KUKA KRL program: MyProgram_029().src

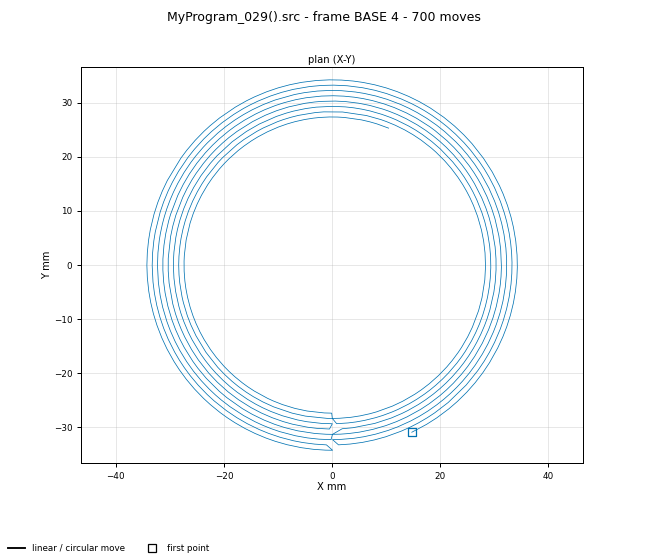
[picture p0: tool path of MyProgram_029().src in frame BASE 4, 700 of 700 moves have a stored position in this frame; points joined in program order, loops and branches not executed]
&ACCESS RVP
&REL 1
&PARAM TEMPLATE = C:\KRC\Roboter\Template\vorgabe
&PARAM EDITMASK = *
DEF MyProgram_029()
; ---- Setting reference (Base) ----
$BASE = BASE_DATA[4]

; --------------------------
; ---- Setting tool (TCP) ----
$TOOL = TOOL_DATA[3]
; --------------------------

$VEL.CP = VEL_APROX_PRINT
Startdeposition()
$VEL.CP = VEL_PRINT
LIN {X 14.7405,Y -30.9266,Z 59,A -69.7461,B 24.853,C -2.7977,E1 25.0726,E2 -567.2107} C_DIS
LIN {X 17.464,Y -29.4746,Z 59,A -65.0615,B 24.8527,C -2.8002,E1 25.084,E2 -571.8873} C_DIS
LIN {X 19.3591,Y -28.2666,Z 59,A -61.3011,B 24.8519,C -2.8074,E1 25.0927,E2 -575.6523} C_DIS
LIN {X 21.5912,Y -26.5997,Z 59,A -56.6338,B 24.8509,C -2.8173,E1 25.103,E2 -580.3259} C_DIS
LIN {X 23.1828,Y -25.2248,Z 59,A -53.0148,B 24.8499,C -2.8266,E1 25.1106,E2 -583.9526} C_DIS
LIN {X 24.9271,Y -23.5028,Z 59,A -49.0912,B 24.8491,C -2.8339,E1 25.1182,E2 -587.8767} C_DIS
LIN {X 26.474,Y -21.7461,Z 59,A -45.15,B 24.848,C -2.8442,E1 25.1254,E2 -591.8243} C_DIS
LIN {X 27.8774,Y -19.9147,Z 59,A -41.382,B 24.8471,C -2.8531,E1 25.1316,E2 -595.5953} C_DIS
LIN {X 29.1256,Y -18.0405,Z 59,A -37.326,B 24.8455,C -2.8677,E1 25.1377,E2 -599.6654} C_DIS
LIN {X 30.6261,Y -15.3561,Z 59,A -32.4503,B 24.8443,C -2.8785,E1 25.1442,E2 -604.541} C_DIS
LIN {X 31.5991,Y -13.2381,Z 59,A -28.9182,B 24.8437,C -2.8846,E1 25.1481,E2 -608.0684} C_DIS
LIN {X 32.2982,Y -11.4269,Z 59,A -25.3896,B 24.8421,C -2.8985,E1 25.1516,E2 -611.6102} C_DIS
LIN {X 32.9807,Y -9.2749,Z 59,A -21.6584,B 24.8409,C -2.9094,E1 25.1545,E2 -615.3459} C_DIS
LIN {X 33.5316,Y -7.0281,Z 59,A -17.8504,B 24.8397,C -2.9205,E1 25.1569,E2 -619.1581} C_DIS
LIN {X 33.9066,Y -4.9084,Z 59,A -14.2291,B 24.8384,C -2.9321,E1 25.1585,E2 -622.7854} C_DIS
LIN {X 34.1715,Y -2.4646,Z 59,A -10.3592,B 24.8374,C -2.9414,E1 25.1595,E2 -626.6544} C_DIS
LIN {X 34.2581,Y -0.4122,Z 59,A -7.0062,B 24.8364,C -2.9509,E1 25.1598,E2 -630.01} C_DIS
LIN {X 34.2094,Y 1.8598,Z 59,A -2.861,B 24.8345,C -2.9678,E1 25.1593,E2 -634.1707} C_DIS
LIN {X 33.9679,Y 4.4635,Z 59,A 1.6751,B 24.8327,C -2.9837,E1 25.1579,E2 -638.7176} C_DIS
LIN {X 33.5424,Y 6.9758,Z 59,A 5.7809,B 24.8315,C -2.9943,E1 25.1558,E2 -642.8245} C_DIS
LIN {X 33.086,Y 8.8916,Z 59,A 8.8785,B 24.8307,C -3.0013,E1 25.1536,E2 -645.9207} C_DIS
LIN {X 32.425,Y 11.062,Z 59,A 12.6485,B 24.8295,C -3.0119,E1 25.1504,E2 -649.6945} C_DIS
LIN {X 31.6198,Y 13.1883,Z 59,A 16.4178,B 24.8283,C -3.0222,E1 25.1465,E2 -653.4673} C_DIS
LIN {X 30.9574,Y 14.6757,Z 59,A 19.4296,B 24.827,C -3.0339,E1 25.1429,E2 -656.4904} C_DIS
LIN {X 29.6029,Y 17.2468,Z 59,A 24.3228,B 24.8255,C -3.0471,E1 25.1362,E2 -661.3895} C_DIS
LIN {X 27.9895,Y 19.7575,Z 59,A 29.8161,B 24.8232,C -3.0665,E1 25.1275,E2 -666.9019} C_DIS
LIN {X 25.8743,Y 22.4561,Z 59,A 34.6343,B 24.8232,C -3.0668,E1 25.119,E2 -671.6983} C_DIS
LIN {X 24.3597,Y 24.0904,Z 59,A 38.3083,B 24.8224,C -3.0739,E1 25.1119,E2 -675.3734} C_DIS
LIN {X 22.6334,Y 25.7185,Z 59,A 42.4549,B 24.8212,C -3.0841,E1 25.1034,E2 -679.5276} C_DIS
LIN {X 20.6758,Y 27.318,Z 59,A 46.7306,B 24.8202,C -3.0922,E1 25.0939,E2 -683.8066} C_DIS
LIN {X 18.1629,Y 29.0492,Z 59,A 51.3273,B 24.8201,C -3.0935,E1 25.0833,E2 -688.3911} C_DIS
LIN {X 16.1457,Y 30.2173,Z 59,A 55.5227,B 24.819,C -3.1026,E1 25.073,E2 -692.5958} C_DIS
LIN {X 14.1516,Y 31.2007,Z 59,A 59.2053,B 24.8186,C -3.1065,E1 25.0637,E2 -696.278} C_DIS
LIN {X 12.0486,Y 32.0715,Z 59,A 62.877,B 24.8183,C -3.1085,E1 25.0542,E2 -699.9463} C_DIS
LIN {X 10.0272,Y 32.7598,Z 59,A 66.5328,B 24.8179,C -3.1123,E1 25.0445,E2 -703.6042} C_DIS
LIN {X 7.884,Y 33.3406,Z 59,A 70.2371,B 24.8176,C -3.1143,E1 25.0345,E2 -707.3078} C_DIS
LIN {X 5.71,Y 33.7808,Z 59,A 73.853,B 24.8176,C -3.1146,E1 25.0246,E2 -710.9203} C_DIS
LIN {X 3.8752,Y 34.0402,Z 59,A 76.9113,B 24.8176,C -3.1147,E1 25.0161,E2 -713.9765} C_DIS
LIN {X 1.7101,Y 34.2177,Z 59,A 80.7532,B 24.8173,C -3.1172,E1 25.0054,E2 -717.8227} C_DIS
LIN {X -0.5043,Y 34.2564,Z 59,A 84.4217,B 24.8174,C -3.1161,E1 24.9951,E2 -721.4883} C_DIS
LIN {X -2.8784,Y 34.1391,Z 59,A 88.2803,B 24.8178,C -3.1132,E1 24.9844,E2 -725.3414} C_DIS
LIN {X -5.6277,Y 33.7946,Z 59,A 93.0032,B 24.818,C -3.1112,E1 24.9714,E2 -730.0635} C_DIS
LIN {X -7.8461,Y 33.3496,Z 59,A 96.8048,B 24.8184,C -3.1082,E1 24.961,E2 -733.8625} C_DIS
LIN {X -9.987,Y 32.772,Z 59,A 100.5274,B 24.8188,C -3.1045,E1 24.951,E2 -737.5822} C_DIS
LIN {X -12.135,Y 32.0388,Z 59,A 104.5504,B 24.8191,C -3.1021,E1 24.9404,E2 -741.6076} C_DIS
LIN {X -14.386,Y 31.0931,Z 59,A 108.4987,B 24.8199,C -3.0948,E1 24.9304,E2 -745.5481} C_DIS
LIN {X -15.8249,Y 30.3861,Z 59,A 111.1524,B 24.8205,C -3.0903,E1 24.9238,E2 -748.1981} C_DIS
LIN {X -17.8874,Y 29.2198,Z 59,A 116.225,B 24.82,C -3.0942,E1 24.9116,E2 -753.2955} C_DIS
LIN {X -20.8096,Y 27.2162,Z 59,A 121.0639,B 24.8226,C -3.0719,E1 24.9008,E2 -758.0982} C_DIS
LIN {X -22.5993,Y 25.7492,Z 59,A 124.3498,B 24.8242,C -3.0581,E1 24.8938,E2 -761.3637} C_DIS
LIN {X -23.6969,Y 24.743,Z 59,A 127.467,B 24.8242,C -3.0581,E1 24.8874,E2 -764.4939} C_DIS
LIN {X -25.329,Y 23.0695,Z 59,A 131.356,B 24.8253,C -3.0486,E1 24.88,E2 -768.3769} C_DIS
LIN {X -26.8917,Y 21.227,Z 59,A 135.0661,B 24.8268,C -3.0354,E1 24.8734,E2 -772.0726} C_DIS
LIN {X -27.957,Y 19.8031,Z 59,A 139.6158,B 24.8261,C -3.0416,E1 24.866,E2 -776.6594} C_DIS
LIN {X -30.4868,Y 15.6302,Z 59,A 146.4974,B 24.83,C -3.0074,E1 24.8565,E2 -783.4949} C_DIS
LIN {X -31.4154,Y 13.6678,Z 59,A 150.3431,B 24.831,C -2.9986,E1 24.8521,E2 -787.3406} C_DIS
LIN {X -32.2494,Y 11.5637,Z 59,A 154.1399,B 24.8323,C -2.9874,E1 24.8483,E2 -791.132} C_DIS
LIN {X -32.9429,Y 9.4083,Z 59,A 157.9699,B 24.8335,C -2.9762,E1 24.8452,E2 -794.9574} C_DIS
LIN {X -33.6357,Y 6.5105,Z 59,A 162.7425,B 24.8355,C -2.959,E1 24.8423,E2 -799.7169} C_DIS
LIN {X -33.9505,Y 4.5959,Z 59,A 166.2829,B 24.8363,C -2.9514,E1 24.8409,E2 -803.2601} C_DIS
LIN {X -34.1811,Y 2.3229,Z 59,A 170.0869,B 24.8376,C -2.9393,E1 24.84,E2 -807.0579} C_DIS
LIN {X -34.2633,Y -0.0539,Z 59,A 174.3256,B 24.8388,C -2.929,E1 24.8398,E2 -811.2976} C_DIS
LIN {X -34.1828,Y -2.2985,Z 59,A 178.423,B 24.8397,C -2.9203,E1 24.8405,E2 -815.3989} C_DIS
LIN {X -33.9145,Y -4.8529,Z 59,A -177.8569,B 24.8417,C -2.9022,E1 24.8418,E2 -819.0978} C_DIS
LIN {X -33.5569,Y -6.905,Z 59,A -174.3787,B 24.8429,C -2.8916,E1 24.8436,E2 -822.5712} C_DIS
LIN {X -33.058,Y -8.9955,Z 59,A -170.6929,B 24.844,C -2.8817,E1 24.8461,E2 -826.2549} C_DIS
LIN {X -32.3999,Y -11.1357,Z 59,A -166.7336,B 24.8449,C -2.8727,E1 24.8496,E2 -830.2152} C_DIS
LIN {X -31.4947,Y -13.4845,Z 59,A -162.6659,B 24.8464,C -2.8597,E1 24.8538,E2 -834.2743} C_DIS
LIN {X -30.5422,Y -15.5218,Z 59,A -158.5503,B 24.8471,C -2.8526,E1 24.8589,E2 -838.3953} C_DIS
LIN {X -29.249,Y -17.8394,Z 59,A -154.637,B 24.8489,C -2.8364,E1 24.8644,E2 -842.2901} C_DIS
LIN {X -28.2742,Y -19.3479,Z 59,A -151.3708,B 24.8494,C -2.8313,E1 24.8695,E2 -845.5605} C_DIS
LIN {X -26.9635,Y -21.1361,Z 59,A -147.6116,B 24.8503,C -2.8231,E1 24.8758,E2 -849.3179} C_DIS
LIN {X -25.4516,Y -22.9341,Z 59,A -143.015,B 24.8505,C -2.8208,E1 24.8843,E2 -853.9298} C_DIS
LIN {X -23.7844,Y -24.6586,Z 59,A -139.5091,B 24.8519,C -2.8077,E1 24.8913,E2 -857.4192} C_DIS
LIN {X -22.5323,Y -25.8077,Z 59,A -136.8285,B 24.8526,C -2.8007,E1 24.8969,E2 -860.0937} C_DIS
LIN {X -20.703,Y -27.2975,Z 59,A -133.39,B 24.8539,C -2.7888,E1 24.9043,E2 -863.5164} C_DIS
LIN {X -19.4209,Y -28.224,Z 59,A -130.7013,B 24.8543,C -2.7849,E1 24.9105,E2 -866.2051} C_DIS
LIN {X -18.0062,Y -29.147,Z 59,A -127.3803,B 24.8543,C -2.7857,E1 24.9183,E2 -869.5387} C_DIS
LIN {X -16.1186,Y -30.2319,Z 59,A -123.6326,B 24.8546,C -2.782,E1 24.9275,E2 -873.2883} C_DIS
LIN {X -14.2682,Y -31.1475,Z 59,A -120.1241,B 24.855,C -2.7787,E1 24.9363,E2 -876.7979} C_DIS
LIN {X -12.2604,Y -31.9911,Z 59,A -116.947,B 24.8559,C -2.7703,E1 24.9445,E2 -879.9618} C_DIS
LIN {X -10.5074,Y -32.6089,Z 59,A -113.4599,B 24.8557,C -2.7719,E1 24.9538,E2 -883.4595} C_DIS
LIN {X -8.3148,Y -33.2357,Z 59,A -109.3423,B 24.8556,C -2.7731,E1 24.9649,E2 -887.586} C_DIS
LIN {X -5.7265,Y -33.7781,Z 59,A -105.2552,B 24.8561,C -2.7677,E1 24.9761,E2 -891.6646} C_DIS
LIN {X -3.4586,Y -34.0851,Z 59,A -101.4077,B 24.8561,C -2.7674,E1 24.9868,E2 -895.514} C_DIS
LIN {X -1.2183,Y -34.2383,Z 59,A -97.6708,B 24.8561,C -2.7674,E1 24.9972,E2 -899.2519} C_DIS
LIN {X 0.0839,Y -34.2576,Z 59,A -95.8071,B 24.8565,C -2.7642,E1 25.0024,E2 -901.108} C_DIS
Enddeposition()
LIN {X 0.0839,Y -34.2576,Z 59,A -95.8071,B 24.8565,C -2.7642,E1 25.0024,E2 -901.108} C_DIS
Startdeposition()
$VEL.CP = VEL_PRINT
LIN {X -1.0513,Y -33.2626,Z 59,A -99.2311,B 24.8565,C -2.7639,E1 24.9928,E2 -897.683} C_DIS
LIN {X -3.2134,Y -33.124,Z 59,A -103.0989,B 24.8567,C -2.7625,E1 24.9821,E2 -893.8101} C_DIS
LIN {X -5.4546,Y -32.8291,Z 59,A -106.4743,B 24.856,C -2.769,E1 24.9728,E2 -890.4474} C_DIS
LIN {X -7.1334,Y -32.5057,Z 59,A -110.1837,B 24.8567,C -2.762,E1 24.9626,E2 -886.7172} C_DIS
LIN {X -9.6035,Y -31.8634,Z 59,A -114.2752,B 24.8561,C -2.7679,E1 24.9516,E2 -882.6331} C_DIS
LIN {X -11.736,Y -31.1412,Z 59,A -117.9092,B 24.8555,C -2.7736,E1 24.942,E2 -879.0056} C_DIS
LIN {X -13.5077,Y -30.4145,Z 59,A -121.0995,B 24.855,C -2.778,E1 24.9338,E2 -875.8184} C_DIS
LIN {X -15.6855,Y -29.3512,Z 59,A -125.7249,B 24.855,C -2.7786,E1 24.9223,E2 -871.1821} C_DIS
LIN {X -17.6429,Y -28.2176,Z 59,A -128.9253,B 24.8537,C -2.7908,E1 24.9146,E2 -868.0009} C_DIS
LIN {X -19.5558,Y -26.9276,Z 59,A -133.4698,B 24.8537,C -2.7917,E1 24.9042,E2 -863.4432} C_DIS
LIN {X -21.821,Y -25.1268,Z 59,A -138.5506,B 24.8528,C -2.7998,E1 24.8932,E2 -858.3625} C_DIS
LIN {X -23.0939,Y -23.962,Z 59,A -141.3685,B 24.852,C -2.807,E1 24.8875,E2 -855.5504} C_DIS
LIN {X -24.7781,Y -22.216,Z 59,A -145.7575,B 24.8512,C -2.814,E1 24.8791,E2 -851.159} C_DIS
LIN {X -26.2348,Y -20.4763,Z 59,A -149.7559,B 24.8504,C -2.8222,E1 24.8721,E2 -847.1614} C_DIS
LIN {X -27.3124,Y -19.0142,Z 59,A -152.9626,B 24.8496,C -2.8291,E1 24.8669,E2 -843.9555} C_DIS
LIN {X -28.269,Y -17.5607,Z 59,A -156.0165,B 24.8489,C -2.8362,E1 24.8624,E2 -840.903} C_DIS
LIN {X -29.1232,Y -16.1048,Z 59,A -158.7971,B 24.848,C -2.8448,E1 24.8586,E2 -838.1285} C_DIS
LIN {X -30.3045,Y -13.7532,Z 59,A -163.3204,B 24.8466,C -2.8572,E1 24.8531,E2 -833.6103} C_DIS
LIN {X -31.1576,Y -11.692,Z 59,A -167.0268,B 24.8453,C -2.8691,E1 24.8493,E2 -829.9117} C_DIS
LIN {X -31.854,Y -9.6343,Z 59,A -170.9227,B 24.8443,C -2.8787,E1 24.846,E2 -826.0166} C_DIS
LIN {X -32.4233,Y -7.4988,Z 59,A -174.8123,B 24.8431,C -2.8894,E1 24.8433,E2 -822.1298} C_DIS
LIN {X -32.8581,Y -5.2808,Z 59,A -178.2301,B 24.8414,C -2.9049,E1 24.8416,E2 -818.7288} C_DIS
LIN {X -33.1309,Y -3.1391,Z 59,A 176.9992,B 24.8411,C -2.9082,E1 24.8402,E2 -813.9373} C_DIS
LIN {X -33.2823,Y -0.0844,Z 59,A 171.9482,B 24.8391,C -2.9262,E1 24.8398,E2 -808.899} C_DIS
LIN {X -33.199,Y 2.3095,Z 59,A 168.1325,B 24.8374,C -2.9415,E1 24.8404,E2 -805.0971} C_DIS
LIN {X -32.9744,Y 4.4963,Z 59,A 164.2866,B 24.8361,C -2.9528,E1 24.8416,E2 -801.2553} C_DIS
LIN {X -32.7069,Y 6.1455,Z 59,A 160.9023,B 24.8356,C -2.9579,E1 24.8433,E2 -797.863} C_DIS
LIN {X -31.8104,Y 9.7779,Z 59,A 155.3438,B 24.8326,C -2.9845,E1 24.8473,E2 -792.336} C_DIS
LIN {X -31.1742,Y 11.6469,Z 59,A 151.4172,B 24.8319,C -2.9906,E1 24.8509,E2 -788.4016} C_DIS
LIN {X -30.3318,Y 13.6925,Z 59,A 147.6169,B 24.8306,C -3.0019,E1 24.8551,E2 -784.6074} C_DIS
LIN {X -29.5573,Y 15.2935,Z 59,A 144.9294,B 24.8293,C -3.0137,E1 24.8585,E2 -781.9336} C_DIS
LIN {X -28.3974,Y 17.352,Z 59,A 139.5884,B 24.8292,C -3.0149,E1 24.8661,E2 -776.5678} C_DIS
LIN {X -26.6676,Y 19.9087,Z 59,A 135.1964,B 24.8267,C -3.0364,E1 24.8732,E2 -772.2059} C_DIS
LIN {X -25.4609,Y 21.4298,Z 59,A 131.4671,B 24.8261,C -3.0417,E1 24.8798,E2 -768.4721} C_DIS
LIN {X -23.7506,Y 23.3114,Z 59,A 127.7417,B 24.8242,C -3.0578,E1 24.8869,E2 -764.7687} C_DIS
LIN {X -22.3273,Y 24.6781,Z 59,A 123.8354,B 24.8238,C -3.0611,E1 24.8948,E2 -760.8544} C_DIS
LIN {X -20.369,Y 26.3176,Z 59,A 119.5644,B 24.8226,C -3.0715,E1 24.9041,E2 -756.5923} C_DIS
LIN {X -18.2065,Y 27.8576,Z 59,A 114.5524,B 24.8221,C -3.0764,E1 24.9156,E2 -751.5751} C_DIS
LIN {X -16.3905,Y 28.9634,Z 59,A 111.5311,B 24.8207,C -3.0886,E1 24.9229,E2 -748.5738} C_DIS
LIN {X -15.1448,Y 29.6333,Z 59,A 109.0401,B 24.8203,C -3.092,E1 24.929,E2 -746.0841} C_DIS
LIN {X -13.7142,Y 30.322,Z 59,A 106.116,B 24.82,C -3.0943,E1 24.9364,E2 -743.1582} C_DIS
LIN {X -11.4232,Y 31.2572,Z 59,A 101.7742,B 24.8194,C -3.0991,E1 24.9477,E2 -738.8185} C_DIS
LIN {X -9.3237,Y 31.9467,Z 59,A 97.9153,B 24.819,C -3.1028,E1 24.958,E2 -734.9618} C_DIS
LIN {X -7.1747,Y 32.4967,Z 59,A 93.6214,B 24.8191,C -3.1015,E1 24.9697,E2 -730.6592} C_DIS
LIN {X -4.1421,Y 33.0205,Z 59,A 88.7457,B 24.8182,C -3.1093,E1 24.9831,E2 -725.7978} C_DIS
LIN {X -1.906,Y 33.2246,Z 59,A 84.9848,B 24.8179,C -3.112,E1 24.9936,E2 -722.0419} C_DIS
LIN {X 0.2942,Y 33.278,Z 59,A 81.1158,B 24.8179,C -3.112,E1 25.0044,E2 -718.1728} C_DIS
LIN {X 2.7961,Y 33.1618,Z 59,A 76.3281,B 24.8185,C -3.1068,E1 25.0178,E2 -713.3749} C_DIS
LIN {X 5.656,Y 32.7955,Z 59,A 71.812,B 24.8181,C -3.1104,E1 25.0302,E2 -708.8715} C_DIS
LIN {X 7.9233,Y 32.3222,Z 59,A 67.8738,B 24.8183,C -3.109,E1 25.0409,E2 -704.9353} C_DIS
LIN {X 10.0959,Y 31.7112,Z 59,A 64.0323,B 24.8185,C -3.1067,E1 25.0512,E2 -701.0951} C_DIS
LIN {X 12.7541,Y 30.7381,Z 59,A 59.1638,B 24.8191,C -3.1022,E1 25.0639,E2 -696.2265} C_DIS
LIN {X 14.6474,Y 29.8823,Z 59,A 55.7532,B 24.8193,C -3.1001,E1 25.0725,E2 -692.8197} C_DIS
LIN {X 15.8991,Y 29.2357,Z 59,A 53.501,B 24.8194,C -3.0991,E1 25.078,E2 -690.5715} C_DIS
LIN {X 17.0583,Y 28.575,Z 59,A 51.1165,B 24.8199,C -3.0948,E1 25.0838,E2 -688.184} C_DIS
LIN {X 18.4365,Y 27.7054,Z 59,A 48.2449,B 24.8205,C -3.0897,E1 25.0905,E2 -685.3096} C_DIS
LIN {X 19.9827,Y 26.612,Z 59,A 45.1035,B 24.821,C -3.0857,E1 25.0976,E2 -682.1699} C_DIS
LIN {X 21.2217,Y 25.6344,Z 59,A 42.3692,B 24.8216,C -3.0806,E1 25.1036,E2 -679.4338} C_DIS
LIN {X 22.8316,Y 24.212,Z 59,A 38.4987,B 24.8227,C -3.0711,E1 25.1116,E2 -675.5565} C_DIS
LIN {X 24.4,Y 22.6311,Z 59,A 34.5848,B 24.8237,C -3.062,E1 25.1191,E2 -671.6377} C_DIS
LIN {X 25.649,Y 21.2048,Z 59,A 31.0911,B 24.8249,C -3.0516,E1 25.1254,E2 -668.1354} C_DIS
LIN {X 27.2532,Y 19.0993,Z 59,A 27.0367,B 24.8254,C -3.0474,E1 25.1321,E2 -664.0905} C_DIS
LIN {X 28.1452,Y 17.7588,Z 59,A 24.4032,B 24.826,C -3.0423,E1 25.1361,E2 -661.4581} C_DIS
LIN {X 28.9934,Y 16.3373,Z 59,A 21.4412,B 24.827,C -3.0333,E1 25.1403,E2 -658.4902} C_DIS
LIN {X 30.0216,Y 14.3599,Z 59,A 16.8708,B 24.8294,C -3.013,E1 25.146,E2 -653.896} C_DIS
LIN {X 31.1351,Y 11.7521,Z 59,A 12.5501,B 24.8301,C -3.0069,E1 25.1505,E2 -649.5848} C_DIS
LIN {X 31.8634,Y 9.6032,Z 59,A 8.7227,B 24.8312,C -2.9966,E1 25.1537,E2 -645.7547} C_DIS
LIN {X 32.3092,Y 7.9769,Z 59,A 5.9432,B 24.832,C -2.9897,E1 25.1557,E2 -642.9749} C_DIS
LIN {X 32.7386,Y 5.9734,Z 59,A 2.5356,B 24.833,C -2.9807,E1 25.1575,E2 -639.5659} C_DIS
LIN {X 33.0211,Y 4.1387,Z 59,A -0.7594,B 24.8343,C -2.9695,E1 25.1588,E2 -636.2639} C_DIS
LIN {X 33.2055,Y 2.2131,Z 59,A -4.0723,B 24.8354,C -2.9595,E1 25.1596,E2 -632.9468} C_DIS
LIN {X 33.276,Y 0.4774,Z 59,A -6.9001,B 24.8362,C -2.9524,E1 25.1598,E2 -630.1191} C_DIS
LIN {X 33.2435,Y -1.5435,Z 59,A -10.5167,B 24.8376,C -2.9396,E1 25.1595,E2 -626.4937} C_DIS
LIN {X 33.0924,Y -3.5208,Z 59,A -14.1374,B 24.8391,C -2.926,E1 25.1585,E2 -622.8622} C_DIS
LIN {X 32.7463,Y -5.9315,Z 59,A -18.1363,B 24.8403,C -2.9157,E1 25.1567,E2 -618.8623} C_DIS
LIN {X 32.2764,Y -8.1086,Z 59,A -21.9835,B 24.8416,C -2.9036,E1 25.1543,E2 -615.0089} C_DIS
LIN {X 31.6616,Y -10.2494,Z 59,A -25.7098,B 24.8427,C -2.8934,E1 25.1513,E2 -611.2798} C_DIS
LIN {X 31.1017,Y -11.8403,Z 59,A -28.5925,B 24.8436,C -2.885,E1 25.1485,E2 -608.3932} C_DIS
LIN {X 30.0639,Y -14.2709,Z 59,A -33.0205,B 24.8449,C -2.8733,E1 25.1434,E2 -603.9616} C_DIS
LIN {X 29.1358,Y -16.0815,Z 59,A -36.4648,B 24.8459,C -2.8641,E1 25.1389,E2 -600.5136} C_DIS
LIN {X 28.1457,Y -17.7579,Z 59,A -39.9421,B 24.8471,C -2.853,E1 25.1339,E2 -597.0278} C_DIS
LIN {X 26.9324,Y -19.5492,Z 59,A -43.682,B 24.8482,C -2.8428,E1 25.1279,E2 -593.282} C_DIS
LIN {X 24.8007,Y -22.1908,Z 59,A -50.4839,B 24.8511,C -2.8152,E1 25.1155,E2 -586.4456} C_DIS
LIN {X 21.4654,Y -25.4313,Z 59,A -58.2661,B 24.8527,C -2.8,E1 25.0994,E2 -578.6588} C_DIS
LIN {X 18.9665,Y -27.3455,Z 59,A -62.2715,B 24.8519,C -2.8074,E1 25.0905,E2 -574.6853} C_DIS
LIN {X 17.5882,Y -28.2518,Z 59,A -65.741,B 24.8534,C -2.7939,E1 25.0823,E2 -571.1951} C_DIS
LIN {X 16.0123,Y -29.1743,Z 59,A -68.4628,B 24.8534,C -2.7939,E1 25.0757,E2 -568.4812} C_DIS
LIN {X 14.5105,Y -29.9489,Z 59,A -71.9666,B 24.8547,C -2.7817,E1 25.0669,E2 -564.958} C_DIS
LIN {X 12.7765,Y -30.7288,Z 59,A -75.3506,B 24.8553,C -2.7756,E1 25.0582,E2 -561.5676} C_DIS
LIN {X 9.9233,Y -31.7653,Z 59,A -80.1944,B 24.8555,C -2.7739,E1 25.0454,E2 -556.7293} C_DIS
LIN {X 7.7788,Y -32.3575,Z 59,A -83.9745,B 24.8558,C -2.7707,E1 25.0352,E2 -552.9472} C_DIS
LIN {X 5.6164,Y -32.8021,Z 59,A -87.8297,B 24.8562,C -2.767,E1 25.0246,E2 -549.0877} C_DIS
LIN {X 3.3246,Y -33.1128,Z 59,A -91.8087,B 24.8564,C -2.7647,E1 25.0135,E2 -545.1061} C_DIS
LIN {X 1.1789,Y -33.2583,Z 59,A -95.4481,B 24.8565,C -2.764,E1 25.0034,E2 -541.4662} C_DIS
LIN {X 1.1789,Y -33.2583,Z 59,A -95.4481,B 24.8565,C -2.764,E1 25.0034,E2 -541.4662} C_DIS
Enddeposition()
LIN {X 0.0782,Y -32.2949,Z 59,A -96.0047,B 24.8532,C -2.7956,E1 25.0021,E2 -540.9851} C_DIS
Startdeposition()
$VEL.CP = VEL_PRINT
LIN {X 1.3776,Y -32.269,Z 59,A -93.085,B 24.8524,C -2.8033,E1 25.0102,E2 -543.9224} C_DIS
LIN {X 4.0439,Y -32.0444,Z 59,A -88.7471,B 24.8526,C -2.8011,E1 25.0223,E2 -548.2523} C_DIS
LIN {X 5.9343,Y -31.7488,Z 59,A -85.0621,B 24.852,C -2.8071,E1 25.0324,E2 -551.9477} C_DIS
LIN {X 8.071,Y -31.2738,Z 59,A -81.2104,B 24.8516,C -2.8105,E1 25.0429,E2 -555.8017} C_DIS
LIN {X 10.3749,Y -30.5864,Z 59,A -77.2542,B 24.8515,C -2.8116,E1 25.0534,E2 -559.7534} C_DIS
LIN {X 12.1046,Y -29.944,Z 59,A -73.5085,B 24.8504,C -2.8219,E1 25.0632,E2 -563.5153} C_DIS
LIN {X 14.5137,Y -28.8539,Z 59,A -69.2101,B 24.8502,C -2.8242,E1 25.074,E2 -567.808} C_DIS
LIN {X 16.12,Y -27.9881,Z 59,A -66.2122,B 24.8499,C -2.8267,E1 25.0814,E2 -570.803} C_DIS
LIN {X 17.7363,Y -26.9929,Z 59,A -62.4207,B 24.8486,C -2.8384,E1 25.0903,E2 -574.6102} C_DIS
LIN {X 19.3678,Y -25.8472,Z 59,A -59.0894,B 24.8482,C -2.8429,E1 25.0979,E2 -577.9403} C_DIS
LIN {X 20.7058,Y -24.7884,Z 59,A -56.1584,B 24.8476,C -2.8481,E1 25.1042,E2 -580.8726} C_DIS
LIN {X 21.9112,Y -23.7297,Z 59,A -53.3433,B 24.847,C -2.8542,E1 25.11,E2 -583.6907} C_DIS
LIN {X 23.0385,Y -22.6368,Z 59,A -50.5791,B 24.8463,C -2.8605,E1 25.1155,E2 -586.4582} C_DIS
LIN {X 24.1384,Y -21.4602,Z 59,A -47.662,B 24.8454,C -2.8683,E1 25.121,E2 -589.381} C_DIS
LIN {X 25.3956,Y -19.9564,Z 59,A -44.4152,B 24.8448,C -2.8741,E1 25.1268,E2 -592.6265} C_DIS
LIN {X 26.4594,Y -18.5229,Z 59,A -40.7136,B 24.8431,C -2.8899,E1 25.1328,E2 -596.3474} C_DIS
LIN {X 27.8025,Y -16.4381,Z 59,A -36.7194,B 24.8424,C -2.8965,E1 25.1387,E2 -600.337} C_DIS
LIN {X 28.8178,Y -14.5852,Z 59,A -32.4602,B 24.8404,C -2.9143,E1 25.1442,E2 -604.6161} C_DIS
LIN {X 29.8223,Y -12.4021,Z 59,A -28.8769,B 24.8401,C -2.9174,E1 25.1483,E2 -608.1871} C_DIS
LIN {X 30.3974,Y -10.9172,Z 59,A -25.7308,B 24.8386,C -2.9304,E1 25.1513,E2 -611.3464} C_DIS
LIN {X 31.0771,Y -8.798,Z 59,A -21.7992,B 24.8373,C -2.9422,E1 25.1545,E2 -615.2835} C_DIS
LIN {X 31.6053,Y -6.6562,Z 59,A -17.8831,B 24.836,C -2.9544,E1 25.1569,E2 -619.2057} C_DIS
LIN {X 32.0568,Y -3.9426,Z 59,A -12.9243,B 24.8341,C -2.9707,E1 25.1589,E2 -624.174} C_DIS
LIN {X 32.2602,Y -1.5811,Z 59,A -8.815,B 24.8328,C -2.9825,E1 25.1597,E2 -628.2868} C_DIS
LIN {X 32.2857,Y 0.9056,Z 59,A -4.4351,B 24.8313,C -2.9959,E1 25.1597,E2 -632.6722} C_DIS
LIN {X 32.1423,Y 3.1738,Z 59,A -0.5081,B 24.8301,C -3.0069,E1 25.1587,E2 -636.602} C_DIS
LIN {X 31.7948,Y 5.6811,Z 59,A 4.3665,B 24.8279,C -3.026,E1 25.1565,E2 -641.4932} C_DIS
LIN {X 31.3644,Y 7.7114,Z 59,A 7.5444,B 24.8274,C -3.0299,E1 25.1545,E2 -644.6621} C_DIS
LIN {X 30.7934,Y 9.7451,Z 59,A 11.3098,B 24.8261,C -3.0412,E1 25.1515,E2 -648.4327} C_DIS
LIN {X 30.0591,Y 11.8168,Z 59,A 15.4478,B 24.8245,C -3.0556,E1 25.1474,E2 -652.5817} C_DIS
LIN {X 28.9876,Y 14.2443,Z 59,A 20.1708,B 24.823,C -3.0687,E1 25.1418,E2 -657.3103} C_DIS
LIN {X 27.5164,Y 16.9133,Z 59,A 25.8446,B 24.8209,C -3.0864,E1 25.1338,E2 -662.9967} C_DIS
LIN {X 26.387,Y 18.6264,Z 59,A 28.9981,B 24.8206,C -3.0887,E1 25.1288,E2 -666.1403} C_DIS
LIN {X 25.0665,Y 20.3681,Z 59,A 32.3439,B 24.8204,C -3.0907,E1 25.1231,E2 -669.4752} C_DIS
LIN {X 23.9611,Y 21.6582,Z 59,A 35.1599,B 24.8199,C -3.0948,E1 25.1179,E2 -672.2882} C_DIS
LIN {X 22.8517,Y 22.8259,Z 59,A 38.5731,B 24.8184,C -3.108,E1 25.1112,E2 -675.7181} C_DIS
LIN {X 20.8232,Y 24.69,Z 59,A 43.6752,B 24.817,C -3.1202,E1 25.1005,E2 -680.8288} C_DIS
LIN {X 19.2896,Y 25.9059,Z 59,A 46.5797,B 24.817,C -3.119,E1 25.0941,E2 -683.7199} C_DIS
LIN {X 17.4983,Y 27.1478,Z 59,A 50.9728,B 24.8156,C -3.1317,E1 25.0839,E2 -688.1284} C_DIS
LIN {X 15.735,Y 28.2064,Z 59,A 54.1304,B 24.8157,C -3.1307,E1 25.0763,E2 -691.2741} C_DIS
LIN {X 14.2471,Y 28.9862,Z 59,A 57.078,B 24.8153,C -3.134,E1 25.069,E2 -694.2216} C_DIS
LIN {X 12.6485,Y 29.7189,Z 59,A 60.8038,B 24.8141,C -3.1446,E1 25.0594,E2 -697.9635} C_DIS
LIN {X 10.1682,Y 30.6561,Z 59,A 65.1234,B 24.8141,C -3.1441,E1 25.0481,E2 -702.2731} C_DIS
LIN {X 8.0767,Y 31.2723,Z 59,A 69.0055,B 24.8138,C -3.1468,E1 25.0376,E2 -706.1553} C_DIS
LIN {X 5.9338,Y 31.7488,Z 59,A 72.9344,B 24.8136,C -3.1489,E1 25.0269,E2 -710.0843} C_DIS
LIN {X 4.3043,Y 32.0105,Z 59,A 75.945,B 24.8134,C -3.1505,E1 25.0185,E2 -713.0961} C_DIS
LIN {X 1.6817,Y 32.2548,Z 59,A 80.4709,B 24.8135,C -3.1491,E1 25.006,E2 -717.6165} C_DIS
LIN {X -0.4578,Y 32.2953,Z 59,A 84.3559,B 24.8135,C -3.1493,E1 24.9951,E2 -721.5018} C_DIS
LIN {X -2.7414,Y 32.1823,Z 59,A 88.9081,B 24.8131,C -3.1528,E1 24.9824,E2 -726.0642} C_DIS
LIN {X -5.1696,Y 31.8824,Z 59,A 92.4827,B 24.8143,C -3.1422,E1 24.9726,E2 -729.6163} C_DIS
LIN {X -6.97,Y 31.5375,Z 59,A 96.5996,B 24.8136,C -3.1482,E1 24.9613,E2 -733.7524} C_DIS
LIN {X -10.5666,Y 30.5214,Z 59,A 102.3808,B 24.8155,C -3.1326,E1 24.9459,E2 -739.5064} C_DIS
LIN {X -12.7308,Y 29.6834,Z 59,A 106.9755,B 24.8156,C -3.1316,E1 24.934,E2 -744.1089} C_DIS
LIN {X -14.7928,Y 28.7119,Z 59,A 110.7428,B 24.8167,C -3.1227,E1 24.9246,E2 -747.8648} C_DIS
LIN {X -16.4195,Y 27.8135,Z 59,A 113.9365,B 24.8174,C -3.1161,E1 24.9169,E2 -751.0523} C_DIS
LIN {X -18.0247,Y 26.8007,Z 59,A 117.6818,B 24.8178,C -3.1132,E1 24.9081,E2 -754.8029} C_DIS
LIN {X -19.6189,Y 25.6574,Z 59,A 121.1288,B 24.8186,C -3.1059,E1 24.9004,E2 -758.2446} C_DIS
LIN {X -21.1497,Y 24.4108,Z 59,A 124.6629,B 24.8195,C -3.0986,E1 24.8929,E2 -761.7749} C_DIS
LIN {X -23.0602,Y 22.6146,Z 59,A 128.7408,B 24.8213,C -3.083,E1 24.8848,E2 -765.8324} C_DIS
LIN {X -23.8783,Y 21.7489,Z 59,A 131.3295,B 24.8214,C -3.0818,E1 24.8799,E2 -768.4297} C_DIS
LIN {X -25.2285,Y 20.1678,Z 59,A 134.6898,B 24.8228,C -3.0698,E1 24.8739,E2 -771.7767} C_DIS
LIN {X -26.1355,Y 18.9774,Z 59,A 137.2737,B 24.8237,C -3.0623,E1 24.8696,E2 -774.3551} C_DIS
LIN {X -27.4017,Y 17.0975,Z 59,A 141.8796,B 24.8244,C -3.0561,E1 24.8625,E2 -778.9693} C_DIS
LIN {X -28.5605,Y 15.0827,Z 59,A 146.0225,B 24.8258,C -3.0445,E1 24.857,E2 -783.1064} C_DIS
LIN {X -29.3531,Y 13.4756,Z 59,A 148.6812,B 24.8273,C -3.0312,E1 24.8538,E2 -785.7477} C_DIS
LIN {X -29.976,Y 12.0266,Z 59,A 151.832,B 24.8279,C -3.0257,E1 24.8504,E2 -788.9028} C_DIS
LIN {X -30.5735,Y 10.4139,Z 59,A 154.8193,B 24.829,C -3.016,E1 24.8477,E2 -791.8839} C_DIS
LIN {X -31.0196,Y 8.9989,Z 59,A 157.4004,B 24.83,C -3.0076,E1 24.8456,E2 -794.4597} C_DIS
LIN {X -31.3982,Y 7.5716,Z 59,A 160.1125,B 24.8308,C -3.0003,E1 24.8437,E2 -797.1701} C_DIS
LIN {X -31.7771,Y 5.7801,Z 59,A 163.1038,B 24.8322,C -2.9882,E1 24.8421,E2 -800.1502} C_DIS
LIN {X -31.969,Y 4.6017,Z 59,A 165.8381,B 24.8324,C -2.9864,E1 24.841,E2 -802.8964} C_DIS
LIN {X -32.2173,Y 2.2913,Z 59,A 169.8768,B 24.8339,C -2.9729,E1 24.84,E2 -806.9269} C_DIS
LIN {X -32.3013,Y -0.0876,Z 59,A 174.4128,B 24.8351,C -2.9621,E1 24.8398,E2 -811.4645} C_DIS
LIN {X -32.1383,Y -3.2137,Z 59,A -179.6026,B 24.8366,C -2.9483,E1 24.8411,E2 -817.4521} C_DIS
LIN {X -31.8021,Y -5.6406,Z 59,A -175.9158,B 24.8387,C -2.9299,E1 24.8428,E2 -821.1166} C_DIS
LIN {X -31.3364,Y -7.8248,Z 59,A -171.8948,B 24.8399,C -2.9185,E1 24.8453,E2 -825.1339} C_DIS
LIN {X -30.5515,Y -10.4786,Z 59,A -167.189,B 24.8417,C -2.9025,E1 24.8492,E2 -829.8287} C_DIS
LIN {X -29.9271,Y -12.1473,Z 59,A -164.009,B 24.8427,C -2.8938,E1 24.8524,E2 -833.0054} C_DIS
LIN {X -29.0225,Y -14.1733,Z 59,A -159.5226,B 24.8433,C -2.8875,E1 24.8578,E2 -837.5013} C_DIS
LIN {X -28.1673,Y -15.805,Z 59,A -156.018,B 24.8441,C -2.8809,E1 24.8625,E2 -841.0085} C_DIS
LIN {X -26.9068,Y -17.8668,Z 59,A -152.0439,B 24.8455,C -2.8675,E1 24.8685,E2 -844.9706} C_DIS
LIN {X -25.6477,Y -19.6315,Z 59,A -148.357,B 24.8466,C -2.857,E1 24.8746,E2 -848.6502} C_DIS
LIN {X -24.1963,Y -21.3953,Z 59,A -144.1664,B 24.8475,C -2.8492,E1 24.8822,E2 -852.8411} C_DIS
LIN {X -22.7591,Y -22.9177,Z 59,A -141.0477,B 24.8489,C -2.8362,E1 24.8883,E2 -855.9421} C_DIS
LIN {X -21.5676,Y -24.0422,Z 59,A -138.06,B 24.8494,C -2.8312,E1 24.8944,E2 -858.9301} C_DIS
LIN {X -20.5169,Y -24.9451,Z 59,A -135.526,B 24.8498,C -2.8274,E1 24.8998,E2 -861.4647} C_DIS
LIN {X -18.882,Y -26.2046,Z 59,A -131.1033,B 24.8498,C -2.8283,E1 24.9098,E2 -865.9053} C_DIS
LIN {X -16.3892,Y -27.8314,Z 59,A -126.3762,B 24.8511,C -2.8153,E1 24.9209,E2 -870.6163} C_DIS
LIN {X -14.2809,Y -28.9697,Z 59,A -121.8492,B 24.8514,C -2.8127,E1 24.9321,E2 -875.1495} C_DIS
LIN {X -12.8899,Y -29.6149,Z 59,A -119.1925,B 24.8518,C -2.8092,E1 24.9389,E2 -877.8042} C_DIS
LIN {X -11.2962,Y -30.2586,Z 59,A -116.5824,B 24.8525,C -2.802,E1 24.9457,E2 -880.4027} C_DIS
LIN {X -9.6591,Y -30.8204,Z 59,A -113.1179,B 24.8523,C -2.8036,E1 24.9549,E2 -883.8776} C_DIS
LIN {X -6.7511,Y -31.5849,Z 59,A -107.2389,B 24.852,C -2.8067,E1 24.9709,E2 -889.7718} C_DIS
LIN {X -4.5659,Y -31.9741,Z 59,A -103.8143,B 24.8527,C -2.8001,E1 24.9803,E2 -893.1838} C_DIS
LIN {X -2.4127,Y -32.2082,Z 59,A -99.9493,B 24.8527,C -2.8001,E1 24.9911,E2 -897.0509} C_DIS
LIN {X -0.1926,Y -32.2979,Z 59,A -96.0166,B 24.8527,C -2.8006,E1 25.002,E2 -900.9851} C_DIS
LIN {X -0.1926,Y -32.2979,Z 59,A -96.0166,B 24.8527,C -2.8006,E1 25.002,E2 -900.9851} C_DIS
Enddeposition()
LIN {X 0.0652,Y -31.3168,Z 59,A -95.9073,B 24.8513,C -2.8137,E1 25.0024,E2 -901.1253} C_DIS
Startdeposition()
$VEL.CP = VEL_PRINT
LIN {X -1.1068,Y -31.2981,Z 59,A -99.6271,B 24.8531,C -2.7965,E1 24.9919,E2 -897.3645} C_DIS
LIN {X -3.1858,Y -31.1553,Z 59,A -103.4462,B 24.8531,C -2.7965,E1 24.9813,E2 -893.5437} C_DIS
LIN {X -6.3199,Y -30.6734,Z 59,A -110.0447,B 24.8537,C -2.7906,E1 24.9631,E2 -886.9243} C_DIS
LIN {X -8.7194,Y -30.0795,Z 59,A -113.6153,B 24.8525,C -2.8025,E1 24.9536,E2 -883.3765} C_DIS
LIN {X -10.6138,Y -29.4643,Z 59,A -117.4725,B 24.8524,C -2.8033,E1 24.9434,E2 -879.514} C_DIS
LIN {X -12.5801,Y -28.68,Z 59,A -121.4455,B 24.8521,C -2.8063,E1 24.9331,E2 -875.539} C_DIS
LIN {X -14.7761,Y -27.6131,Z 59,A -125.116,B 24.8507,C -2.8189,E1 24.924,E2 -871.8889} C_DIS
LIN {X -16.6113,Y -26.5492,Z 59,A -130.2465,B 24.8513,C -2.8133,E1 24.9117,E2 -866.7293} C_DIS
LIN {X -19.4806,Y -24.5216,Z 59,A -136.4341,B 24.8499,C -2.8262,E1 24.8978,E2 -860.5505} C_DIS
LIN {X -20.8515,Y -23.3669,Z 59,A -140.4746,B 24.8499,C -2.8262,E1 24.8894,E2 -856.4939} C_DIS
LIN {X -23.2562,Y -20.9752,Z 59,A -145.624,B 24.8476,C -2.8478,E1 24.8795,E2 -851.3738} C_DIS
LIN {X -24.8198,Y -19.0991,Z 59,A -150.152,B 24.8466,C -2.8576,E1 24.8716,E2 -846.848} C_DIS
LIN {X -25.7802,Y -17.7817,Z 59,A -153.0554,B 24.8457,C -2.8654,E1 24.8669,E2 -843.9491} C_DIS
LIN {X -27.3493,Y -15.2582,Z 59,A -157.8136,B 24.8437,C -2.8846,E1 24.86,E2 -839.2123} C_DIS
LIN {X -28.1335,Y -13.7587,Z 59,A -161.7987,B 24.8435,C -2.8861,E1 24.8549,E2 -835.2095} C_DIS
LIN {X -28.9543,Y -11.9346,Z 59,A -165.2704,B 24.8422,C -2.8977,E1 24.8511,E2 -831.7463} C_DIS
LIN {X -29.6203,Y -10.1706,Z 59,A -169.7188,B 24.8419,C -2.9003,E1 24.847,E2 -827.279} C_DIS
LIN {X -30.3821,Y -7.5981,Z 59,A -173.9,B 24.8398,C -2.92,E1 24.8439,E2 -823.1207} C_DIS
LIN {X -30.8937,Y -5.1344,Z 59,A -178.3414,B 24.8381,C -2.9351,E1 24.8416,E2 -818.6892} C_DIS
LIN {X -31.1611,Y -3.1292,Z 59,A 177.7518,B 24.837,C -2.945,E1 24.8403,E2 -814.7827} C_DIS
LIN {X -31.3034,Y -0.9353,Z 59,A 173.5454,B 24.8358,C -2.9562,E1 24.8398,E2 -810.5778} C_DIS
LIN {X -31.298,Y 1.1104,Z 59,A 169.9872,B 24.8343,C -2.9692,E1 24.84,E2 -807.0292} C_DIS
LIN {X -31.1064,Y 3.6314,Z 59,A 165.2399,B 24.8328,C -2.9828,E1 24.8412,E2 -802.286} C_DIS
LIN {X -30.7754,Y 5.8022,Z 59,A 161.0463,B 24.8315,C -2.994,E1 24.8432,E2 -798.0944} C_DIS
LIN {X -30.2298,Y 8.1823,Z 59,A 157.1409,B 24.8295,C -3.0118,E1 24.8458,E2 -794.2087} C_DIS
LIN {X -29.8743,Y 9.3982,Z 59,A 153.7615,B 24.8295,C -3.0113,E1 24.8486,E2 -790.8087} C_DIS
LIN {X -28.5429,Y 12.888,Z 59,A 148.2538,B 24.8262,C -3.0411,E1 24.8543,E2 -785.3416} C_DIS
LIN {X -27.5475,Y 14.8973,Z 59,A 142.9271,B 24.8258,C -3.0439,E1 24.8611,E2 -779.9932} C_DIS
LIN {X -26.4073,Y 16.8347,Z 59,A 139.2031,B 24.8242,C -3.0581,E1 24.8665,E2 -776.2842} C_DIS
LIN {X -25.0108,Y 18.8484,Z 59,A 134.6658,B 24.8229,C -3.0696,E1 24.8739,E2 -771.7521} C_DIS
LIN {X -23.4372,Y 20.7723,Z 59,A 130.2372,B 24.8214,C -3.0819,E1 24.8819,E2 -767.3327} C_DIS
LIN {X -22.1252,Y 22.1646,Z 59,A 126.6804,B 24.8205,C -3.0897,E1 24.8888,E2 -763.7794} C_DIS
LIN {X -20.8764,Y 23.3447,Z 59,A 123.4869,B 24.8197,C -3.0964,E1 24.8954,E2 -760.5891} C_DIS
LIN {X -19.1496,Y 24.7809,Z 59,A 120.0848,B 24.8181,C -3.1108,E1 24.9027,E2 -757.2086} C_DIS
LIN {X -17.9269,Y 25.6792,Z 59,A 116.8711,B 24.8178,C -3.1127,E1 24.91,E2 -753.9882} C_DIS
LIN {X -16.2109,Y 26.7957,Z 59,A 112.4627,B 24.8177,C -3.114,E1 24.9205,E2 -749.569} C_DIS
LIN {X -14.162,Y 27.9326,Z 59,A 108.6026,B 24.8164,C -3.1247,E1 24.9299,E2 -745.7235} C_DIS
LIN {X -12.501,Y 28.7138,Z 59,A 105.3231,B 24.8158,C -3.1303,E1 24.9383,E2 -742.4494} C_DIS
LIN {X -10.4546,Y 29.5212,Z 59,A 101.0982,B 24.8154,C -3.1336,E1 24.9493,E2 -738.2237} C_DIS
LIN {X -8.8896,Y 30.029,Z 59,A 98.0458,B 24.815,C -3.1366,E1 24.9575,E2 -735.1731} C_DIS
LIN {X -6.7653,Y 30.5784,Z 59,A 94.203,B 24.8144,C -3.1418,E1 24.9679,E2 -731.3375} C_DIS
LIN {X -4.8541,Y 30.9393,Z 59,A 89.541,B 24.8153,C -3.134,E1 24.9808,E2 -726.6524} C_DIS
LIN {X -1.9637,Y 31.2564,Z 59,A 85.1186,B 24.814,C -3.145,E1 24.993,E2 -722.2543} C_DIS
LIN {X 0.2067,Y 31.317,Z 59,A 81.0236,B 24.814,C -3.1447,E1 25.0044,E2 -718.1584} C_DIS
LIN {X 2.1962,Y 31.2403,Z 59,A 77.6104,B 24.8138,C -3.1471,E1 25.0139,E2 -714.7522} C_DIS
LIN {X 4.0972,Y 31.0486,Z 59,A 74.3228,B 24.8136,C -3.1486,E1 25.023,E2 -711.4708} C_DIS
LIN {X 5.7617,Y 30.7832,Z 59,A 71.348,B 24.8136,C -3.1488,E1 25.0312,E2 -708.4993} C_DIS
LIN {X 7.459,Y 30.4165,Z 59,A 67.7584,B 24.8143,C -3.1427,E1 25.041,E2 -704.9003} C_DIS
LIN {X 9.5841,Y 29.8152,Z 59,A 63.7698,B 24.8146,C -3.1404,E1 25.0517,E2 -700.9132} C_DIS
LIN {X 11.4971,Y 29.1308,Z 59,A 60.2593,B 24.8146,C -3.1393,E1 25.0608,E2 -697.4076} C_DIS
LIN {X 13.7486,Y 28.1384,Z 59,A 55.4226,B 24.8157,C -3.1304,E1 25.0731,E2 -692.5621} C_DIS
LIN {X 15.6124,Y 27.1486,Z 59,A 51.42,B 24.8165,C -3.1236,E1 25.0829,E2 -688.555} C_DIS
LIN {X 18.0141,Y 25.6186,Z 59,A 46.9896,B 24.8165,C -3.1247,E1 25.0932,E2 -684.1419} C_DIS
LIN {X 19.0101,Y 24.8876,Z 59,A 43.9854,B 24.8179,C -3.1119,E1 25.0999,E2 -681.1182} C_DIS
LIN {X 21.2564,Y 22.9995,Z 59,A 39.1899,B 24.8183,C -3.1087,E1 25.11,E2 -676.3339} C_DIS
LIN {X 22.5343,Y 21.7486,Z 59,A 35.3118,B 24.82,C -3.0944,E1 25.1176,E2 -672.4384} C_DIS
LIN {X 23.6978,Y 20.4751,Z 59,A 32.168,B 24.8208,C -3.0875,E1 25.1234,E2 -669.2925} C_DIS
LIN {X 25.362,Y 18.3734,Z 59,A 27.8714,B 24.8212,C -3.0836,E1 25.1307,E2 -665.0071} C_DIS
LIN {X 26.2742,Y 17.0437,Z 59,A 24.9788,B 24.822,C -3.077,E1 25.1352,E2 -662.1132} C_DIS
LIN {X 26.9691,Y 15.9206,Z 59,A 22.7233,B 24.8225,C -3.0729,E1 25.1384,E2 -659.8594} C_DIS
LIN {X 27.6424,Y 14.7212,Z 59,A 20.2156,B 24.8232,C -3.0664,E1 25.1418,E2 -657.3493} C_DIS
LIN {X 28.629,Y 12.6955,Z 59,A 15.3129,B 24.8257,C -3.0449,E1 25.1476,E2 -652.4223} C_DIS
LIN {X 29.4639,Y 10.6148,Z 59,A 11.616,B 24.8264,C -3.0385,E1 25.1513,E2 -648.7309} C_DIS
LIN {X 30.1229,Y 8.5678,Z 59,A 7.6857,B 24.8278,C -3.0271,E1 25.1544,E2 -644.7958} C_DIS
LIN {X 30.8485,Y 5.4016,Z 59,A 0.9591,B 24.831,C -2.9988,E1 25.1582,E2 -638.0414} C_DIS
LIN {X 31.1741,Y 2.9974,Z 59,A -3.1557,B 24.832,C -2.9894,E1 25.1594,E2 -633.9288} C_DIS
LIN {X 31.3164,Y -0.3515,Z 59,A -8.3722,B 24.8328,C -2.9826,E1 25.1597,E2 -628.7271} C_DIS
LIN {X 31.2448,Y -2.1334,Z 59,A -11.5106,B 24.8338,C -2.974,E1 25.1593,E2 -625.5871} C_DIS
LIN {X 31.1128,Y -3.5764,Z 59,A -14.387,B 24.835,C -2.9627,E1 25.1585,E2 -622.7009} C_DIS
LIN {X 30.8727,Y -5.2614,Z 59,A -18.2338,B 24.8372,C -2.9431,E1 25.1567,E2 -618.8305} C_DIS
LIN {X 30.3592,Y -7.6895,Z 59,A -22.1848,B 24.8379,C -2.937,E1 25.1542,E2 -614.8877} C_DIS
LIN {X 29.75,Y -9.784,Z 59,A -26.4573,B 24.8397,C -2.9211,E1 25.1506,E2 -610.6018} C_DIS
LIN {X 28.9339,Y -11.9841,Z 59,A -30.5466,B 24.8408,C -2.911,E1 25.1464,E2 -606.5113} C_DIS
LIN {X 27.7817,Y -14.456,Z 59,A -35.6543,B 24.8425,C -2.8949,E1 25.1401,E2 -601.3929} C_DIS
LIN {X 26.3436,Y -16.9355,Z 59,A -40.7288,B 24.8439,C -2.8826,E1 25.1328,E2 -596.315} C_DIS
LIN {X 25.0677,Y -18.7725,Z 59,A -44.6171,B 24.8448,C -2.8743,E1 25.1264,E2 -592.426} C_DIS
LIN {X 23.9789,Y -20.1451,Z 59,A -47.7514,B 24.8456,C -2.867,E1 25.1209,E2 -589.2889} C_DIS
LIN {X 22.4364,Y -21.8495,Z 59,A -51.8533,B 24.8465,C -2.8581,E1 25.113,E2 -585.1839} C_DIS
LIN {X 21.1269,Y -23.1182,Z 59,A -55.2964,B 24.8475,C -2.8491,E1 25.106,E2 -581.7334} C_DIS
LIN {X 19.9339,Y -24.1547,Z 59,A -58.5315,B 24.8486,C -2.8385,E1 25.0991,E2 -578.4856} C_DIS
LIN {X 17.9733,Y -25.647,Z 59,A -62.607,B 24.849,C -2.8347,E1 25.0899,E2 -574.4156} C_DIS
LIN {X 16.3366,Y -26.7192,Z 59,A -66.4531,B 24.8501,C -2.8248,E1 25.0808,E2 -570.5583} C_DIS
LIN {X 13.837,Y -28.095,Z 59,A -71.3324,B 24.8506,C -2.8202,E1 25.0687,E2 -565.6819} C_DIS
LIN {X 11.892,Y -28.9717,Z 59,A -75.2928,B 24.8513,C -2.8139,E1 25.0586,E2 -561.7161} C_DIS
LIN {X 9.907,Y -29.7089,Z 59,A -79.4107,B 24.8521,C -2.8062,E1 25.0477,E2 -557.5883} C_DIS
LIN {X 7.5467,Y -30.3949,Z 59,A -83.7265,B 24.8523,C -2.8036,E1 25.0361,E2 -553.2732} C_DIS
LIN {X 5.0797,Y -30.9031,Z 59,A -88.2448,B 24.8526,C -2.8009,E1 25.0237,E2 -548.7536} C_DIS
LIN {X 3.0101,Y -31.1727,Z 59,A -91.7893,B 24.8526,C -2.8017,E1 25.0138,E2 -545.2136} C_DIS
LIN {X 1.5768,Y -31.2782,Z 59,A -94.4581,B 24.8527,C -2.8002,E1 25.0064,E2 -542.5422} C_DIS
LIN {X 0.0652,Y -31.3168,Z 59,A -95.9071,B 24.8513,C -2.8136,E1 25.0024,E2 -541.1253} C_DIS
Enddeposition()
LIN {X 0.0652,Y -31.3168,Z 59,A -95.9071,B 24.8513,C -2.8136,E1 25.0024,E2 -541.1253} C_DIS
Startdeposition()
$VEL.CP = VEL_PRINT
LIN {X 1.8608,Y -30.2801,Z 59,A -92.0548,B 24.8488,C -2.8365,E1 25.0133,E2 -545.031} C_DIS
LIN {X 3.8672,Y -30.0894,Z 59,A -87.6755,B 24.8479,C -2.8451,E1 25.0255,E2 -549.4274} C_DIS
LIN {X 7.9042,Y -29.2891,Z 59,A -79.9875,B 24.8473,C -2.8513,E1 25.0464,E2 -557.1194} C_DIS
LIN {X 10.9225,Y -28.3026,Z 59,A -74.6858,B 24.8473,C -2.8507,E1 25.0604,E2 -562.409} C_DIS
LIN {X 12.8928,Y -27.4609,Z 59,A -71.0034,B 24.8471,C -2.8523,E1 25.0697,E2 -566.0863} C_DIS
LIN {X 14.0481,Y -26.8878,Z 59,A -68.15,B 24.8462,C -2.8613,E1 25.0769,E2 -568.9532} C_DIS
LIN {X 16.0002,Y -25.7746,Z 59,A -64.254,B 24.8458,C -2.8647,E1 25.0862,E2 -572.8451} C_DIS
LIN {X 17.2727,Y -24.9396,Z 59,A -61.304,B 24.8451,C -2.8711,E1 25.0931,E2 -575.8006} C_DIS
LIN {X 18.6975,Y -23.8903,Z 59,A -58.1163,B 24.8446,C -2.8761,E1 25.1002,E2 -578.9886} C_DIS
LIN {X 19.9311,Y -22.871,Z 59,A -54.8915,B 24.8436,C -2.8853,E1 25.107,E2 -582.2226} C_DIS
LIN {X 21.0757,Y -21.8208,Z 59,A -52.2182,B 24.8432,C -2.8888,E1 25.1125,E2 -584.8932} C_DIS
LIN {X 22.189,Y -20.688,Z 59,A -49.0109,B 24.8421,C -2.8987,E1 25.1187,E2 -588.11} C_DIS
LIN {X 23.4187,Y -19.285,Z 59,A -45.6234,B 24.8413,C -2.9058,E1 25.1248,E2 -591.499} C_DIS
LIN {X 24.3561,Y -18.0866,Z 59,A -42.7938,B 24.8406,C -2.9128,E1 25.1296,E2 -594.3317} C_DIS
LIN {X 25.256,Y -16.807,Z 59,A -39.6986,B 24.8395,C -2.9226,E1 25.1345,E2 -597.4349} C_DIS
LIN {X 26.1271,Y -15.4176,Z 59,A -36.8165,B 24.8389,C -2.9284,E1 25.1387,E2 -600.3161} C_DIS
LIN {X 26.7497,Y -14.3108,Z 59,A -34.5797,B 24.8383,C -2.9331,E1 25.1417,E2 -602.5523} C_DIS
LIN {X 27.5143,Y -12.7785,Z 59,A -30.7978,B 24.8365,C -2.9498,E1 25.1463,E2 -606.3534} C_DIS
LIN {X 28.2069,Y -11.1671,Z 59,A -27.9868,B 24.8361,C -2.953,E1 25.1492,E2 -609.1564} C_DIS
LIN {X 28.6803,Y -9.8875,Z 59,A -24.902,B 24.8345,C -2.9675,E1 25.1521,E2 -612.2583} C_DIS
LIN {X 29.1802,Y -8.2974,Z 59,A -21.2087,B 24.8326,C -2.9845,E1 25.155,E2 -615.9707} C_DIS
LIN {X 29.9214,Y -5.004,Z 59,A -15.8964,B 24.832,C -2.9899,E1 25.1579,E2 -621.2649} C_DIS
LIN {X 30.1728,Y -3.151,Z 59,A -12.8043,B 24.8314,C -2.9951,E1 25.159,E2 -624.3509} C_DIS
LIN {X 30.3234,Y -0.9056,Z 59,A -8.3798,B 24.8296,C -3.0107,E1 25.1597,E2 -628.7862} C_DIS
LIN {X 30.3162,Y 1.1209,Z 59,A -3.7703,B 24.8271,C -3.0331,E1 25.1595,E2 -633.4214} C_DIS
LIN {X 30.1514,Y 3.3496,Z 59,A 0.7367,B 24.8251,C -3.05,E1 25.1582,E2 -637.9416} C_DIS
LIN {X 29.578,Y 6.7428,Z 59,A 6.6199,B 24.8238,C -3.0614,E1 25.1551,E2 -643.8175} C_DIS
LIN {X 29.0137,Y 8.8621,Z 59,A 10.7233,B 24.8225,C -3.0731,E1 25.152,E2 -647.925} C_DIS
LIN {X 28.4498,Y 10.5324,Z 59,A 13.7029,B 24.8219,C -3.0781,E1 25.1492,E2 -650.8996} C_DIS
LIN {X 27.6625,Y 12.4544,Z 59,A 18.4141,B 24.8194,C -3.0993,E1 25.1439,E2 -655.6354} C_DIS
LIN {X 26.3395,Y 15.0519,Z 59,A 23.281,B 24.8187,C -3.1056,E1 25.1375,E2 -660.4917} C_DIS
LIN {X 25.5062,Y 16.4246,Z 59,A 26.0587,B 24.8181,C -3.11,E1 25.1334,E2 -663.2659} C_DIS
LIN {X 24.8075,Y 17.4626,Z 59,A 28.3033,B 24.8176,C -3.1143,E1 25.1299,E2 -665.5096} C_DIS
LIN {X 23.9629,Y 18.6043,Z 59,A 31.5707,B 24.816,C -3.128,E1 25.1243,E2 -668.794} C_DIS
LIN {X 22.4548,Y 20.3994,Z 59,A 35.6474,B 24.8154,C -3.1335,E1 25.1168,E2 -672.8652} C_DIS
LIN {X 21.1057,Y 21.7918,Z 59,A 39.1672,B 24.8147,C -3.1393,E1 25.1099,E2 -676.384} C_DIS
LIN {X 19.8567,Y 22.935,Z 59,A 42.2837,B 24.8141,C -3.1445,E1 25.1034,E2 -679.5004} C_DIS
LIN {X 18.6872,Y 23.8979,Z 59,A 45.7124,B 24.8127,C -3.1565,E1 25.0959,E2 -682.9445} C_DIS
LIN {X 17.3011,Y 24.9199,Z 59,A 48.6431,B 24.8125,C -3.158,E1 25.0892,E2 -685.8687} C_DIS
LIN {X 15.7255,Y 25.9424,Z 59,A 52.4106,B 24.8115,C -3.1658,E1 25.0803,E2 -689.6428} C_DIS
LIN {X 13.6683,Y 27.0833,Z 59,A 56.5141,B 24.8113,C -3.1676,E1 25.0702,E2 -693.739} C_DIS
LIN {X 12.0526,Y 27.84,Z 59,A 59.5864,B 24.8113,C -3.168,E1 25.0624,E2 -696.8045} C_DIS
LIN {X 10.5791,Y 28.4323,Z 59,A 62.6354,B 24.8109,C -3.1715,E1 25.0545,E2 -699.8549} C_DIS
LIN {X 9.4037,Y 28.8427,Z 59,A 65.763,B 24.8096,C -3.1818,E1 25.0461,E2 -703.0013} C_DIS
LIN {X 6.9635,Y 29.5271,Z 59,A 70.1465,B 24.8098,C -3.1803,E1 25.0343,E2 -707.3745} C_DIS
LIN {X 4.9005,Y 29.9387,Z 59,A 74.2816,B 24.8094,C -3.1834,E1 25.0229,E2 -711.5125} C_DIS
LIN {X 2.5085,Y 30.2329,Z 59,A 78.5067,B 24.8097,C -3.1807,E1 25.0112,E2 -715.7282} C_DIS
LIN {X 0.5924,Y 30.3309,Z 59,A 82.7128,B 24.8091,C -3.1862,E1 24.9994,E2 -719.9465} C_DIS
LIN {X -1.9474,Y 30.2745,Z 59,A 86.6979,B 24.8102,C -3.1767,E1 24.9884,E2 -723.9097} C_DIS
LIN {X -3.2076,Y 30.1667,Z 59,A 89.0011,B 24.8105,C -3.1747,E1 24.982,E2 -726.2094} C_DIS
LIN {X -4.98,Y 29.9254,Z 59,A 93.4161,B 24.8096,C -3.1823,E1 24.9698,E2 -730.6464} C_DIS
LIN {X -8.0652,Y 29.2451,Z 59,A 99.121,B 24.8105,C -3.1743,E1 24.9543,E2 -736.3401} C_DIS
LIN {X -10.2782,Y 28.5427,Z 59,A 102.538,B 24.8122,C -3.1605,E1 24.9453,E2 -739.7306} C_DIS
LIN {X -12.3524,Y 27.7082,Z 59,A 108.5623,B 24.811,C -3.1704,E1 24.9298,E2 -745.7925} C_DIS
LIN {X -14.7158,Y 26.5289,Z 59,A 113.1577,B 24.8124,C -3.1588,E1 24.9185,E2 -750.373} C_DIS
LIN {X -17.6046,Y 24.7061,Z 59,A 118.9885,B 24.8144,C -3.1415,E1 24.905,E2 -756.1816} C_DIS
LIN {X -19.1069,Y 23.5637,Z 59,A 122.1579,B 24.8157,C -3.1309,E1 24.8981,E2 -759.3374} C_DIS
LIN {X -20.2824,Y 22.56,Z 59,A 125.4372,B 24.8161,C -3.1273,E1 24.8912,E2 -762.621} C_DIS
LIN {X -21.5187,Y 21.3841,Z 59,A 128.5419,B 24.8171,C -3.1189,E1 24.885,E2 -765.7187} C_DIS
LIN {X -22.5677,Y 20.2739,Z 59,A 131.347,B 24.818,C -3.1113,E1 24.8797,E2 -768.5179} C_DIS
LIN {X -23.797,Y 18.8157,Z 59,A 135.4986,B 24.8186,C -3.1063,E1 24.8724,E2 -772.6769} C_DIS
LIN {X -25.1523,Y 16.9615,Z 59,A 139.2049,B 24.8205,C -3.0901,E1 24.8664,E2 -776.3624} C_DIS
LIN {X -25.9395,Y 15.7311,Z 59,A 142.2136,B 24.8212,C -3.0843,E1 24.862,E2 -779.3727} C_DIS
LIN {X -26.8542,Y 14.1128,Z 59,A 146.1374,B 24.822,C -3.0774,E1 24.8567,E2 -783.3007} C_DIS
LIN {X -27.6282,Y 12.5304,Z 59,A 150.091,B 24.8226,C -3.0723,E1 24.8521,E2 -787.2636} C_DIS
LIN {X -28.9019,Y 9.2203,Z 59,A 155.9311,B 24.8256,C -3.0459,E1 24.8467,E2 -793.0738} C_DIS
LIN {X -29.4686,Y 7.2064,Z 59,A 160.1922,B 24.8267,C -3.036,E1 24.8436,E2 -797.3359} C_DIS
LIN {X -29.8732,Y 5.2846,Z 59,A 164.527,B 24.8275,C -3.029,E1 24.8415,E2 -801.6795} C_DIS
LIN {X -30.3111,Y 1.2515,Z 59,A 171.0845,B 24.8312,C -2.9972,E1 24.8399,E2 -808.2002} C_DIS
LIN {X -30.3186,Y -1.0537,Z 59,A 176.4775,B 24.8319,C -2.991,E1 24.8401,E2 -813.6108} C_DIS
LIN {X -30.1509,Y -3.3536,Z 59,A -179.0238,B 24.8333,C -2.9786,E1 24.8414,E2 -818.1068} C_DIS
LIN {X -29.4736,Y -7.1858,Z 59,A -172.5271,B 24.8364,C -2.9502,E1 24.8449,E2 -824.574} C_DIS
LIN {X -28.9651,Y -9.0193,Z 59,A -168.7462,B 24.8375,C -2.9411,E1 24.8479,E2 -828.3547} C_DIS
LIN {X -28.4371,Y -10.5665,Z 59,A -165.936,B 24.8387,C -2.9302,E1 24.8505,E2 -831.1549} C_DIS
LIN {X -27.9062,Y -11.8986,Z 59,A -163.1507,B 24.8394,C -2.9232,E1 24.8535,E2 -833.9388} C_DIS
LIN {X -27.271,Y -13.289,Z 59,A -159.7528,B 24.8399,C -2.9191,E1 24.8576,E2 -837.3455} C_DIS
LIN {X -25.9937,Y -15.6421,Z 59,A -154.4445,B 24.8411,C -2.9079,E1 24.8649,E2 -842.6547} C_DIS
LIN {X -24.7417,Y -17.5552,Z 59,A -150.1715,B 24.8423,C -2.897,E1 24.8717,E2 -846.9227} C_DIS
LIN {X -22.8327,Y -19.975,Z 59,A -145.0121,B 24.8443,C -2.8785,E1 24.8808,E2 -852.0617} C_DIS
LIN {X -21.2666,Y -21.6349,Z 59,A -139.8728,B 24.8446,C -2.8763,E1 24.8908,E2 -857.2178} C_DIS
LIN {X -19.2705,Y -23.4307,Z 59,A -135.3086,B 24.846,C -2.8625,E1 24.9005,E2 -861.7669} C_DIS
LIN {X -17.3251,Y -24.9032,Z 59,A -130.2195,B 24.8464,C -2.8591,E1 24.912,E2 -866.8656} C_DIS
LIN {X -14.9659,Y -26.3888,Z 59,A -125.5575,B 24.8478,C -2.8462,E1 24.9231,E2 -871.5112} C_DIS
LIN {X -13.1041,Y -27.3606,Z 59,A -121.5859,B 24.8483,C -2.8415,E1 24.933,E2 -875.4823} C_DIS
LIN {X -11.091,Y -28.2368,Z 59,A -117.1607,B 24.8485,C -2.84,E1 24.9444,E2 -879.9138} C_DIS
LIN {X -9.0399,Y -28.9588,Z 59,A -113.0381,B 24.8488,C -2.8369,E1 24.9553,E2 -884.0369} C_DIS
LIN {X -7.335,Y -29.4366,Z 59,A -109.3961,B 24.8487,C -2.838,E1 24.9652,E2 -887.6866} C_DIS
LIN {X -4.5324,Y -29.9966,Z 59,A -104.6887,B 24.8496,C -2.8293,E1 24.9781,E2 -892.3782} C_DIS
LIN {X -2.819,Y -30.2057,Z 59,A -101.0248,B 24.8492,C -2.833,E1 24.9883,E2 -896.0532} C_DIS
LIN {X -0.4913,Y -30.3323,Z 59,A -96.6276,B 24.8492,C -2.8335,E1 25.0006,E2 -900.4523} C_DIS
LIN {X -0.4913,Y -30.3323,Z 59,A -96.6276,B 24.8492,C -2.8335,E1 25.0006,E2 -900.4523} C_DIS
Enddeposition()
LIN {X 0.0409,Y -29.3539,Z 59,A -96.8614,B 24.8487,C -2.8379,E1 24.9999,E2 -900.229} C_DIS
Startdeposition()
$VEL.CP = VEL_PRINT
LIN {X -1.9496,Y -29.2914,Z 59,A -102.0979,B 24.8501,C -2.8244,E1 24.9852,E2 -894.959} C_DIS
LIN {X -4.7352,Y -28.9719,Z 59,A -106.8504,B 24.8493,C -2.8322,E1 24.9721,E2 -890.2216} C_DIS
LIN {X -6.4354,Y -28.6419,Z 59,A -110.6418,B 24.8496,C -2.8299,E1 24.9618,E2 -886.4201} C_DIS
LIN {X -9.1522,Y -27.893,Z 59,A -115.8967,B 24.8489,C -2.8358,E1 24.9477,E2 -881.1705} C_DIS
LIN {X -11.3101,Y -27.0897,Z 59,A -120.3108,B 24.8484,C -2.8407,E1 24.9362,E2 -876.7584} C_DIS
LIN {X -12.8893,Y -26.3751,Z 59,A -123.5131,B 24.8478,C -2.846,E1 24.9282,E2 -873.5608} C_DIS
LIN {X -14.1799,Y -25.7047,Z 59,A -126.3059,B 24.8474,C -2.85,E1 24.9213,E2 -870.7697} C_DIS
LIN {X -15.6462,Y -24.8392,Z 59,A -130.0856,B 24.8473,C -2.851,E1 24.9123,E2 -866.9807} C_DIS
LIN {X -17.5749,Y -23.514,Z 59,A -134.7859,B 24.8466,C -2.8575,E1 24.9016,E2 -862.2795} C_DIS
LIN {X -18.9092,Y -22.4555,Z 59,A -137.5623,B 24.8455,C -2.8677,E1 24.8956,E2 -859.517} C_DIS
LIN {X -20.1567,Y -21.3423,Z 59,A -141.1067,B 24.845,C -2.8719,E1 24.8883,E2 -855.9684} C_DIS
LIN {X -21.5029,Y -19.9857,Z 59,A -144.4846,B 24.8439,C -2.8824,E1 24.8818,E2 -852.6009} C_DIS
LIN {X -22.4689,Y -18.8932,Z 59,A -147.6902,B 24.8435,C -2.886,E1 24.8759,E2 -849.3894} C_DIS
LIN {X -23.4296,Y -17.6873,Z 59,A -150.8069,B 24.8428,C -2.8923,E1 24.8706,E2 -846.2729} C_DIS
LIN {X -24.3221,Y -16.4384,Z 59,A -154.2919,B 24.8424,C -2.8962,E1 24.8651,E2 -842.78} C_DIS
LIN {X -25.9007,Y -13.8189,Z 59,A -159.8678,B 24.8404,C -2.9144,E1 24.8574,E2 -837.2186} C_DIS
LIN {X -26.616,Y -12.3844,Z 59,A -162.9723,B 24.8394,C -2.9231,E1 24.8537,E2 -834.1181} C_DIS
LIN {X -27.4376,Y -10.4383,Z 59,A -166.8,B 24.8379,C -2.9367,E1 24.8497,E2 -830.3015} C_DIS
LIN {X -27.9631,Y -8.9365,Z 59,A -170.1223,B 24.8371,C -2.9442,E1 24.8467,E2 -826.9783} C_DIS
LIN {X -28.3393,Y -7.6592,Z 59,A -172.8456,B 24.8363,C -2.951,E1 24.8447,E2 -824.2555} C_DIS
LIN {X -28.946,Y -4.8904,Z 59,A -179.1963,B 24.8351,C -2.9625,E1 24.8413,E2 -817.8947} C_DIS
LIN {X -29.253,Y -2.4625,Z 59,A 176.4531,B 24.8331,C -2.9799,E1 24.8401,E2 -813.5597} C_DIS
LIN {X -29.3549,Y -0.3332,Z 59,A 173.208,B 24.831,C -2.9987,E1 24.8398,E2 -810.3401} C_DIS
LIN {X -29.3365,Y 1.074,Z 59,A 170.4583,B 24.83,C -3.0072,E1 24.8399,E2 -807.5943} C_DIS
LIN {X -29.2559,Y 2.4179,Z 59,A 166.8035,B 24.8298,C -3.0089,E1 24.8407,E2 -803.9214} C_DIS
LIN {X -28.9084,Y 5.1081,Z 59,A 162.1296,B 24.8275,C -3.0293,E1 24.8426,E2 -799.2687} C_DIS
LIN {X -28.6227,Y 6.5206,Z 59,A 159.0833,B 24.8267,C -3.0365,E1 24.8444,E2 -796.2217} C_DIS
LIN {X -28.1643,Y 8.2799,Z 59,A 155.6119,B 24.8254,C -3.0479,E1 24.8469,E2 -792.7573} C_DIS
LIN {X -27.4552,Y 10.3921,Z 59,A 150.5514,B 24.8244,C -3.0563,E1 24.8517,E2 -787.6884} C_DIS
LIN {X -26.6494,Y 12.3126,Z 59,A 147.3404,B 24.8224,C -3.0738,E1 24.8553,E2 -784.5016} C_DIS
LIN {X -25.6132,Y 14.3439,Z 59,A 141.6576,B 24.8219,C -3.0783,E1 24.8628,E2 -778.7995} C_DIS
LIN {X -24.2707,Y 16.5143,Z 59,A 136.919,B 24.8201,C -3.0934,E1 24.87,E2 -774.0733} C_DIS
LIN {X -22.5234,Y 18.8264,Z 59,A 132.1122,B 24.8177,C -3.1139,E1 24.8783,E2 -769.2927} C_DIS
LIN {X -21.3,Y 20.2017,Z 59,A 127.1934,B 24.8177,C -3.1132,E1 24.8877,E2 -764.3508} C_DIS
LIN {X -18.5134,Y 22.7824,Z 59,A 120.7225,B 24.815,C -3.1364,E1 24.9012,E2 -757.9098} C_DIS
LIN {X -15.8616,Y 24.7021,Z 59,A 113.2931,B 24.8145,C -3.1409,E1 24.9183,E2 -750.4662} C_DIS
LIN {X -13.4849,Y 26.0757,Z 59,A 108.1707,B 24.8132,C -3.1516,E1 24.9309,E2 -745.3547} C_DIS
LIN {X -10.3292,Y 27.479,Z 59,A 102.2939,B 24.8113,C -3.1679,E1 24.9459,E2 -739.5035} C_DIS
LIN {X -8.4973,Y 28.0994,Z 59,A 98.8228,B 24.8105,C -3.1747,E1 24.9551,E2 -736.0425} C_DIS
LIN {X -7.124,Y 28.4784,Z 59,A 95.7956,B 24.8104,C -3.1754,E1 24.9633,E2 -733.0123} C_DIS
LIN {X -4.8968,Y 28.9448,Z 59,A 90.4406,B 24.8109,C -3.1708,E1 24.978,E2 -727.6406} C_DIS
LIN {X -2.9557,Y 29.207,Z 59,A 87.4284,B 24.8098,C -3.1801,E1 24.9863,E2 -724.6487} C_DIS
LIN {X 0.0587,Y 29.356,Z 59,A 80.6062,B 24.8106,C -3.1732,E1 25.0054,E2 -717.8092} C_DIS
LIN {X 2.4193,Y 29.2564,Z 59,A 77.1276,B 24.8094,C -3.184,E1 25.015,E2 -714.3576} C_DIS
LIN {X 4.0103,Y 29.0812,Z 59,A 73.599,B 24.8099,C -3.1794,E1 25.0248,E2 -710.8209} C_DIS
LIN {X 5.4978,Y 28.8366,Z 59,A 70.9876,B 24.8096,C -3.1816,E1 25.032,E2 -708.2177} C_DIS
LIN {X 7.0215,Y 28.5042,Z 59,A 67.1799,B 24.8107,C -3.1724,E1 25.0424,E2 -704.3933} C_DIS
LIN {X 9.2209,Y 27.8703,Z 59,A 63.3249,B 24.8104,C -3.1753,E1 25.0526,E2 -700.5523} C_DIS
LIN {X 10.8095,Y 27.2937,Z 59,A 60.2887,B 24.8104,C -3.1751,E1 25.0605,E2 -697.5219} C_DIS
LIN {X 11.8629,Y 26.8525,Z 59,A 57.4351,B 24.8115,C -3.166,E1 25.0679,E2 -694.6538} C_DIS
LIN {X 14.16,Y 25.7157,Z 59,A 53.34,B 24.8111,C -3.1696,E1 25.078,E2 -690.5785} C_DIS
LIN {X 15.4442,Y 24.9656,Z 59,A 49.9117,B 24.8123,C -3.1597,E1 25.0863,E2 -687.1371} C_DIS
LIN {X 16.763,Y 24.0995,Z 59,A 47.2266,B 24.8123,C -3.1592,E1 25.0925,E2 -684.46} C_DIS
LIN {X 18.4353,Y 22.8458,Z 59,A 42.1121,B 24.8146,C -3.1404,E1 25.1038,E2 -679.3195} C_DIS
LIN {X 20.0244,Y 21.4668,Z 59,A 37.7878,B 24.8158,C -3.1298,E1 25.1127,E2 -674.9877} C_DIS
LIN {X 22.298,Y 19.0942,Z 59,A 32.1406,B 24.8164,C -3.1249,E1 25.1233,E2 -669.3538} C_DIS
LIN {X 23.6268,Y 17.4232,Z 59,A 28.3473,B 24.817,C -3.1195,E1 25.1298,E2 -665.5657} C_DIS
LIN {X 24.4155,Y 16.2998,Z 59,A 25.2865,B 24.8183,C -3.1083,E1 25.1346,E2 -662.4935} C_DIS
LIN {X 25.4572,Y 14.619,Z 59,A 21.6296,B 24.8192,C -3.1009,E1 25.1398,E2 -658.8376} C_DIS
LIN {X 26.0614,Y 13.5129,Z 59,A 19.0891,B 24.8201,C -3.0933,E1 25.1431,E2 -656.2926} C_DIS
LIN {X 26.7599,Y 12.07,Z 59,A 16.0141,B 24.821,C -3.0854,E1 25.1467,E2 -653.2155} C_DIS
LIN {X 27.683,Y 9.7694,Z 59,A 11.4157,B 24.8223,C -3.0746,E1 25.1514,E2 -648.6172} C_DIS
LIN {X 28.2303,Y 8.0522,Z 59,A 7.3598,B 24.8243,C -3.0576,E1 25.1546,E2 -644.544} C_DIS
LIN {X 28.7514,Y 5.9273,Z 59,A 3.2601,B 24.8255,C -3.0469,E1 25.1571,E2 -640.4428} C_DIS
LIN {X 29.1416,Y 3.5441,Z 59,A -1.2026,B 24.8268,C -3.0357,E1 25.1589,E2 -635.9798} C_DIS
LIN {X 29.3126,Y 1.5976,Z 59,A -4.9137,B 24.828,C -3.0252,E1 25.1596,E2 -632.2659} C_DIS
LIN {X 29.3524,Y -0.4736,Z 59,A -9.2359,B 24.8298,C -3.009,E1 25.1596,E2 -627.9311} C_DIS
LIN {X 29.2567,Y -2.4143,Z 59,A -12.8328,B 24.8309,C -2.9996,E1 25.159,E2 -624.3333} C_DIS
LIN {X 29.0646,Y -4.127,Z 59,A -15.7796,B 24.8315,C -2.9944,E1 25.158,E2 -621.3916} C_DIS
LIN {X 28.7532,Y -5.9192,Z 59,A -19.8917,B 24.8335,C -2.9762,E1 25.1558,E2 -617.2605} C_DIS
LIN {X 28.3589,Y -7.586,Z 59,A -22.8659,B 24.8342,C -2.9706,E1 25.1538,E2 -614.2902} C_DIS
LIN {X 27.8542,Y -9.269,Z 59,A -25.9442,B 24.8348,C -2.9647,E1 25.1512,E2 -611.2153} C_DIS
LIN {X 27.2754,Y -10.8555,Z 59,A -29.8096,B 24.8367,C -2.9476,E1 25.1473,E2 -607.3309} C_DIS
LIN {X 26.5531,Y -12.5188,Z 59,A -32.8753,B 24.8372,C -2.9431,E1 25.1438,E2 -604.2713} C_DIS
LIN {X 25.7894,Y -14.0246,Z 59,A -36.5922,B 24.8389,C -2.9284,E1 25.139,E2 -600.5391} C_DIS
LIN {X 24.6495,Y -15.9435,Z 59,A -40.4589,B 24.8395,C -2.9224,E1 25.1333,E2 -596.678} C_DIS
LIN {X 23.9673,Y -16.952,Z 59,A -42.744,B 24.8401,C -2.9171,E1 25.1297,E2 -594.3915} C_DIS
LIN {X 23.0691,Y -18.155,Z 59,A -46.319,B 24.8418,C -2.9015,E1 25.1236,E2 -590.7965} C_DIS
LIN {X 21.4909,Y -19.9987,Z 59,A -50.6581,B 24.8426,C -2.8946,E1 25.1155,E2 -586.4604} C_DIS
LIN {X 20.3778,Y -21.1312,Z 59,A -53.6399,B 24.8432,C -2.8887,E1 25.1096,E2 -583.4772} C_DIS
LIN {X 19.1748,Y -22.2289,Z 59,A -56.8579,B 24.844,C -2.8811,E1 25.1029,E2 -580.254} C_DIS
LIN {X 18.0908,Y -23.1198,Z 59,A -59.4117,B 24.8444,C -2.8775,E1 25.0973,E2 -577.7012} C_DIS
LIN {X 17.0955,Y -23.8648,Z 59,A -61.8055,B 24.8449,C -2.8729,E1 25.0919,E2 -575.3051} C_DIS
LIN {X 15.6633,Y -24.8285,Z 59,A -65.3878,B 24.8459,C -2.8641,E1 25.0835,E2 -571.7135} C_DIS
LIN {X 14.2633,Y -25.6577,Z 59,A -68.804,B 24.8468,C -2.8558,E1 25.0752,E2 -568.288} C_DIS
LIN {X 12.1588,Y -26.7198,Z 59,A -72.8324,B 24.8468,C -2.855,E1 25.0651,E2 -564.2683} C_DIS
LIN {X 11.1208,Y -27.1681,Z 59,A -75.3932,B 24.8476,C -2.8479,E1 25.0585,E2 -561.6967} C_DIS
LIN {X 9.4059,Y -27.8077,Z 59,A -78.6301,B 24.8477,C -2.8471,E1 25.05,E2 -558.4645} C_DIS
LIN {X 8.046,Y -28.232,Z 59,A -81.8867,B 24.8486,C -2.8389,E1 25.0413,E2 -555.194} C_DIS
LIN {X 5.9924,Y -28.738,Z 59,A -85.8735,B 24.8488,C -2.8366,E1 25.0304,E2 -551.2072} C_DIS
LIN {X 4.4237,Y -29.021,Z 59,A -88.7936,B 24.8488,C -2.8363,E1 25.0224,E2 -548.2894} C_DIS
LIN {X 2.937,Y -29.2089,Z 59,A -92.0179,B 24.8494,C -2.8315,E1 25.0134,E2 -545.0561} C_DIS
LIN {X 0.8412,Y -29.3439,Z 59,A -95.6281,B 24.849,C -2.8349,E1 25.0034,E2 -541.455} C_DIS
LIN {X 0.8412,Y -29.3439,Z 59,A -95.6281,B 24.849,C -2.8349,E1 25.0034,E2 -541.455} C_DIS
Enddeposition()
LIN {X 0.0354,Y -28.372,Z 59,A -96.4583,B 24.8464,C -2.8589,E1 25.0012,E2 -540.6821} C_DIS
Startdeposition()
$VEL.CP = VEL_PRINT
LIN {X 1.3557,Y -28.3428,Z 59,A -93.0499,B 24.8456,C -2.8671,E1 25.0108,E2 -544.1092} C_DIS
LIN {X 3.4761,Y -28.1618,Z 59,A -89.0055,B 24.8456,C -2.8669,E1 25.022,E2 -548.1504} C_DIS
LIN {X 5.1782,Y -27.8992,Z 59,A -85.2843,B 24.845,C -2.872,E1 25.0323,E2 -551.8799} C_DIS
LIN {X 6.9419,Y -27.5132,Z 59,A -81.6529,B 24.8447,C -2.8753,E1 25.0421,E2 -555.514} C_DIS
LIN {X 8.2237,Y -27.1573,Z 59,A -78.4773,B 24.8438,C -2.8836,E1 25.0507,E2 -558.7037} C_DIS
LIN {X 11.1393,Y -26.0976,Z 59,A -73.4107,B 24.8443,C -2.8788,E1 25.0638,E2 -563.7479} C_DIS
LIN {X 13.0409,Y -25.201,Z 59,A -67.8451,B 24.8419,C -2.9003,E1 25.0778,E2 -569.3497} C_DIS
LIN {X 15.3258,Y -23.8806,Z 59,A -63.527,B 24.8422,C -2.8983,E1 25.0881,E2 -573.6497} C_DIS
LIN {X 16.5024,Y -23.083,Z 59,A -60.5484,B 24.8414,C -2.9053,E1 25.0949,E2 -576.6345} C_DIS
LIN {X 17.9799,Y -21.9523,Z 59,A -56.3188,B 24.8399,C -2.9188,E1 25.1042,E2 -580.8803} C_DIS
LIN {X 19.6876,Y -20.4343,Z 59,A -51.9811,B 24.8391,C -2.926,E1 25.1131,E2 -585.2175} C_DIS
LIN {X 21.2105,Y -18.8491,Z 59,A -48.2312,B 24.8388,C -2.9285,E1 25.1202,E2 -588.957} C_DIS
LIN {X 22.2282,Y -17.6373,Z 59,A -44.245,B 24.8369,C -2.9463,E1 25.1273,E2 -592.967} C_DIS
LIN {X 23.3368,Y -16.1419,Z 59,A -41.0753,B 24.8366,C -2.9491,E1 25.1325,E2 -596.1278} C_DIS
LIN {X 23.9392,Y -15.234,Z 59,A -38.3882,B 24.8352,C -2.9612,E1 25.1365,E2 -598.83} C_DIS
LIN {X 25.0697,Y -13.292,Z 59,A -33.9936,B 24.834,C -2.9723,E1 25.1425,E2 -603.228} C_DIS
LIN {X 25.9437,Y -11.4926,Z 59,A -29.3607,B 24.8318,C -2.9916,E1 25.1479,E2 -607.8816} C_DIS
LIN {X 27.0918,Y -8.438,Z 59,A -23.581,B 24.8307,C -3.0012,E1 25.1533,E2 -613.6515} C_DIS
LIN {X 27.7224,Y -6.0522,Z 59,A -17.9068,B 24.828,C -3.0253,E1 25.157,E2 -619.3501} C_DIS
LIN {X 28.2409,Y -2.7592,Z 59,A -11.3747,B 24.8258,C -3.0438,E1 25.1594,E2 -625.8874} C_DIS
LIN {X 28.3747,Y -0.2908,Z 59,A -6.7908,B 24.8247,C -3.0541,E1 25.1598,E2 -630.4685} C_DIS
LIN {X 28.2868,Y 2.2404,Z 59,A -1.2458,B 24.8222,C -3.0755,E1 25.1589,E2 -636.0312} C_DIS
LIN {X 28.0291,Y 4.4203,Z 59,A 2.3838,B 24.8218,C -3.0789,E1 25.1575,E2 -639.6474} C_DIS
LIN {X 27.6254,Y 6.4798,Z 59,A 7.6544,B 24.8188,C -3.1047,E1 25.1543,E2 -644.9485} C_DIS
LIN {X 26.9102,Y 9.0005,Z 59,A 12.4191,B 24.8177,C -3.1135,E1 25.1503,E2 -649.7069} C_DIS
LIN {X 26.133,Y 11.0558,Z 59,A 16.3309,B 24.817,C -3.1195,E1 25.1463,E2 -653.6113} C_DIS
LIN {X 25.4868,Y 12.4733,Z 59,A 19.2896,B 24.8163,C -3.1258,E1 25.1428,E2 -656.569} C_DIS
LIN {X 24.8914,Y 13.6229,Z 59,A 21.9537,B 24.8154,C -3.1333,E1 25.1393,E2 -659.237} C_DIS
LIN {X 24.1724,Y 14.862,Z 59,A 25.0336,B 24.8142,C -3.143,E1 25.1348,E2 -662.3241} C_DIS
LIN {X 23.2612,Y 16.2507,Z 59,A 28.6404,B 24.8129,C -3.1543,E1 25.1292,E2 -665.9399} C_DIS
LIN {X 22.0379,Y 17.8742,Z 59,A 32.2385,B 24.8125,C -3.1579,E1 25.123,E2 -669.5295} C_DIS
LIN {X 20.7979,Y 19.3034,Z 59,A 36.6797,B 24.8106,C -3.1735,E1 25.1147,E2 -673.9881} C_DIS
LIN {X 19.1853,Y 20.9067,Z 59,A 40.5654,B 24.8105,C -3.1746,E1 25.1069,E2 -677.8602} C_DIS
LIN {X 18.3809,Y 21.6172,Z 59,A 43.2654,B 24.8093,C -3.1848,E1 25.1011,E2 -680.5738} C_DIS
LIN {X 16.4671,Y 23.1084,Z 59,A 47.6882,B 24.8089,C -3.1878,E1 25.0913,E2 -684.9878} C_DIS
LIN {X 14.9642,Y 24.109,Z 59,A 51.5967,B 24.8079,C -3.1963,E1 25.0821,E2 -688.9037} C_DIS
LIN {X 13.4303,Y 24.9959,Z 59,A 55.1549,B 24.8073,C -3.2008,E1 25.0734,E2 -692.4624} C_DIS
LIN {X 11.6728,Y 25.8632,Z 59,A 58.9713,B 24.8069,C -3.2039,E1 25.0637,E2 -696.2763} C_DIS
LIN {X 10.0437,Y 26.5383,Z 59,A 62.2194,B 24.8069,C -3.2041,E1 25.0553,E2 -699.5176} C_DIS
LIN {X 9.0343,Y 26.8988,Z 59,A 65.0555,B 24.8059,C -3.2128,E1 25.0478,E2 -702.3687} C_DIS
LIN {X 6.3416,Y 27.6577,Z 59,A 71.6802,B 24.8043,C -3.2259,E1 25.0298,E2 -709.0148} C_DIS
LIN {X 1.9388,Y 28.3091,Z 59,A 80.252,B 24.8046,C -3.2232,E1 25.0061,E2 -717.5741} C_DIS
LIN {X -1.5339,Y 28.3339,Z 59,A 86.3415,B 24.8059,C -3.2128,E1 24.9891,E2 -723.6392} C_DIS
LIN {X -3.1189,Y 28.2029,Z 59,A 90.2971,B 24.8053,C -3.2179,E1 24.9781,E2 -727.6093} C_DIS
LIN {X -6.1993,Y 27.69,Z 59,A 95.7188,B 24.8068,C -3.2053,E1 24.9633,E2 -733.0068} C_DIS
LIN {X -7.6686,Y 27.3194,Z 59,A 98.6194,B 24.8073,C -3.201,E1 24.9555,E2 -735.9013} C_DIS
LIN {X -9.1082,Y 26.8739,Z 59,A 101.7336,B 24.8076,C -3.1981,E1 24.9472,E2 -739.0143} C_DIS
LIN {X -10.1451,Y 26.4998,Z 59,A 104.7978,B 24.8072,C -3.2021,E1 24.9392,E2 -742.0945} C_DIS
LIN {X -12.7338,Y 25.3576,Z 59,A 109.7576,B 24.8089,C -3.1876,E1 24.9267,E2 -747.0319} C_DIS
LIN {X -13.9338,Y 24.7188,Z 59,A 113.2278,B 24.8088,C -3.1886,E1 24.9182,E2 -750.5146} C_DIS
LIN {X -16.3084,Y 23.2202,Z 59,A 118.4264,B 24.8105,C -3.1744,E1 24.9061,E2 -755.6963} C_DIS
LIN {X -17.607,Y 22.2521,Z 59,A 122.6193,B 24.8105,C -3.1744,E1 24.8969,E2 -759.9047} C_DIS
LIN {X -20.2706,Y 19.856,Z 59,A 129.0581,B 24.8132,C -3.1522,E1 24.8838,E2 -766.3167} C_DIS
LIN {X -21.1102,Y 18.961,Z 59,A 132.3146,B 24.8132,C -3.1516,E1 24.8778,E2 -769.5863} C_DIS
LIN {X -23.2051,Y 16.3308,Z 59,A 138.3915,B 24.8159,C -3.129,E1 24.8675,E2 -775.6381} C_DIS
LIN {X -24.0995,Y 14.9794,Z 59,A 141.387,B 24.8172,C -3.1182,E1 24.863,E2 -778.623} C_DIS
LIN {X -24.9373,Y 13.5387,Z 59,A 145.1358,B 24.818,C -3.1113,E1 24.8579,E2 -782.3748} C_DIS
LIN {X -25.7892,Y 11.8357,Z 59,A 148.9131,B 24.8194,C -3.0997,E1 24.8534,E2 -786.1448} C_DIS
LIN {X -26.5667,Y 9.9687,Z 59,A 153.2929,B 24.8206,C -3.0895,E1 24.8489,E2 -790.5247} C_DIS
LIN {X -27.1579,Y 8.2223,Z 59,A 156.5667,B 24.8222,C -3.0753,E1 24.8461,E2 -793.7833} C_DIS
LIN {X -27.5845,Y 6.6531,Z 59,A 160.1891,B 24.8231,C -3.0674,E1 24.8436,E2 -797.408} C_DIS
LIN {X -27.9437,Y 4.9315,Z 59,A 163.513,B 24.8246,C -3.0549,E1 24.8419,E2 -800.7216} C_DIS
LIN {X -28.158,Y 3.501,Z 59,A 166.5706,B 24.8255,C -3.0467,E1 24.8407,E2 -803.7778} C_DIS
LIN {X -28.3294,Y 1.6137,Z 59,A 170.2662,B 24.827,C -3.0339,E1 24.8399,E2 -807.465} C_DIS
LIN {X -28.3788,Y 0.0146,Z 59,A 173.9377,B 24.8278,C -3.0266,E1 24.8399,E2 -811.1411} C_DIS
LIN {X -28.3195,Y -1.7847,Z 59,A 177.1311,B 24.8294,C -3.0126,E1 24.8402,E2 -814.32} C_DIS
LIN {X -28.1841,Y -3.2893,Z 59,A -179.14,B 24.83,C -3.0076,E1 24.8413,E2 -818.0593} C_DIS
LIN {X -27.7608,Y -5.8738,Z 59,A -174.5795,B 24.8323,C -2.9868,E1 24.8436,E2 -822.5971} C_DIS
LIN {X -27.5132,Y -6.9423,Z 59,A -171.6847,B 24.8326,C -2.9847,E1 24.8456,E2 -825.5038} C_DIS
LIN {X -26.7791,Y -9.3832,Z 59,A -167.4016,B 24.8349,C -2.964,E1 24.8491,E2 -829.7619} C_DIS
LIN {X -26.1518,Y -11.0112,Z 59,A -162.868,B 24.8352,C -2.9609,E1 24.8539,E2 -834.3133} C_DIS
LIN {X -25.1727,Y -13.0957,Z 59,A -157.6869,B 24.8362,C -2.952,E1 24.8604,E2 -839.5011} C_DIS
LIN {X -23.3377,Y -16.1406,Z 59,A -150.3955,B 24.8381,C -2.9349,E1 24.8715,E2 -846.7882} C_DIS
LIN {X -21.1649,Y -18.9001,Z 59,A -144.153,B 24.8406,C -2.9126,E1 24.8825,E2 -853.0062} C_DIS
LIN {X -19.8596,Y -20.2676,Z 59,A -140.2948,B 24.8414,C -2.905,E1 24.8901,E2 -856.8628} C_DIS
LIN {X -18.5463,Y -21.4759,Z 59,A -136.9467,B 24.8424,C -2.8962,E1 24.8971,E2 -860.2031} C_DIS
LIN {X -17.3639,Y -22.4423,Z 59,A -133.6207,B 24.8428,C -2.8926,E1 24.9044,E2 -863.5329} C_DIS
LIN {X -15.9094,Y -23.4959,Z 59,A -130.0231,B 24.8434,C -2.8866,E1 24.9126,E2 -867.1284} C_DIS
LIN {X -14.5736,Y -24.3468,Z 59,A -126.7757,B 24.8439,C -2.8824,E1 24.9203,E2 -870.3758} C_DIS
LIN {X -12.8178,Y -25.3154,Z 59,A -122.7561,B 24.8445,C -2.877,E1 24.9302,E2 -874.3938} C_DIS
LIN {X -10.7867,Y -26.2449,Z 59,A -117.5843,B 24.8444,C -2.8781,E1 24.9435,E2 -879.5803} C_DIS
LIN {X -7.3956,Y -27.3947,Z 59,A -109.9736,B 24.8445,C -2.8765,E1 24.9639,E2 -887.2002} C_DIS
LIN {X -4.939,Y -27.9423,Z 59,A -104.9316,B 24.8448,C -2.8743,E1 24.9777,E2 -892.2423} C_DIS
LIN {X -0.9438,Y -28.3598,Z 59,A -98.0559,B 24.8461,C -2.8621,E1 24.9968,E2 -899.0921} C_DIS
LIN {X 0.0354,Y -28.372,Z 59,A -96.4581,B 24.8464,C -2.8589,E1 25.0012,E2 -900.6821} C_DIS
Enddeposition()
LIN {X 0.0354,Y -28.372,Z 59,A -96.4581,B 24.8464,C -2.8589,E1 25.0012,E2 -900.6821} C_DIS
Startdeposition()
$VEL.CP = VEL_PRINT
LIN {X -0.0754,Y -27.3946,Z 59,A -97.5071,B 24.8455,C -2.868,E1 24.9983,E2 -899.655} C_DIS
LIN {X -1.4417,Y -27.3565,Z 59,A -101.459,B 24.8465,C -2.8579,E1 24.9872,E2 -895.6781} C_DIS
LIN {X -4.6267,Y -27.0013,Z 59,A -107.0925,B 24.8454,C -2.8685,E1 24.9717,E2 -890.0656} C_DIS
LIN {X -6.8835,Y -26.5158,Z 59,A -113.1906,B 24.8463,C -2.8602,E1 24.9551,E2 -883.9396} C_DIS
LIN {X -9.1733,Y -25.8131,Z 59,A -117.3452,B 24.8451,C -2.871,E1 24.9441,E2 -879.803} C_DIS
LIN {X -10.8766,Y -25.1425,Z 59,A -120.6533,B 24.8443,C -2.8789,E1 24.9356,E2 -876.5064} C_DIS
LIN {X -11.95,Y -24.651,Z 59,A -124.256,B 24.8449,C -2.8729,E1 24.9265,E2 -872.8801} C_DIS
LIN {X -14.3762,Y -23.3194,Z 59,A -129.4979,B 24.8436,C -2.8849,E1 24.9138,E2 -867.6514} C_DIS
LIN {X -15.6401,Y -22.4911,Z 59,A -132.2772,B 24.8428,C -2.8927,E1 24.9074,E2 -864.8813} C_DIS
LIN {X -16.5769,Y -21.8101,Z 59,A -135.1872,B 24.8428,C -2.8933,E1 24.9009,E2 -861.9621} C_DIS
LIN {X -17.9946,Y -20.6558,Z 59,A -138.7339,B 24.8417,C -2.9022,E1 24.8933,E2 -858.4234} C_DIS
LIN {X -19.0477,Y -19.6889,Z 59,A -141.6053,B 24.841,C -2.909,E1 24.8875,E2 -855.5563} C_DIS
LIN {X -20.0101,Y -18.71,Z 59,A -144.529,B 24.8404,C -2.9146,E1 24.8818,E2 -852.6335} C_DIS
LIN {X -21.404,Y -17.0977,Z 59,A -149.9677,B 24.84,C -2.9182,E1 24.8721,E2 -847.1782} C_DIS
LIN {X -22.4932,Y -15.6372,Z 59,A -153.4736,B 24.8387,C -2.9294,E1 24.8665,E2 -843.6818} C_DIS
LIN {X -23.6826,Y -13.7682,Z 59,A -157.5057,B 24.837,C -2.945,E1 24.8606,E2 -839.6664} C_DIS
LIN {X -24.4532,Y -12.3495,Z 59,A -161.3539,B 24.8363,C -2.951,E1 24.8556,E2 -835.8122} C_DIS
LIN {X -25.1719,Y -10.8087,Z 59,A -164.5029,B 24.835,C -2.9634,E1 24.8521,E2 -832.6754} C_DIS
LIN {X -25.7267,Y -9.4131,Z 59,A -167.4986,B 24.8339,C -2.9731,E1 24.8491,E2 -829.6863} C_DIS
LIN {X -26.2672,Y -7.7778,Z 59,A -171.673,B 24.8331,C -2.9802,E1 24.8456,E2 -825.5048} C_DIS
LIN {X -26.7462,Y -5.9253,Z 59,A -175.5642,B 24.8317,C -2.9928,E1 24.843,E2 -821.6209} C_DIS
LIN {X -27.0526,Y -4.3157,Z 59,A -178.9447,B 24.8305,C -3.0034,E1 24.8414,E2 -818.2458} C_DIS
LIN {X -27.2352,Y -2.951,Z 59,A 178.0164,B 24.8296,C -3.0113,E1 24.8404,E2 -815.2077} C_DIS
LIN {X -27.3711,Y -1.1356,Z 59,A 174.3071,B 24.8281,C -3.0237,E1 24.8398,E2 -811.5058} C_DIS
LIN {X -27.3852,Y 0.7185,Z 59,A 170.7419,B 24.8266,C -3.0376,E1 24.8398,E2 -807.9524} C_DIS
LIN {X -27.3371,Y 1.7764,Z 59,A 167.6299,B 24.8264,C -3.0394,E1 24.8404,E2 -804.8258} C_DIS
LIN {X -26.9983,Y 4.6452,Z 59,A 161.123,B 24.8245,C -3.0556,E1 24.8431,E2 -798.319} C_DIS
LIN {X -26.2794,Y 7.7369,Z 59,A 155.2522,B 24.8216,C -3.0803,E1 24.8472,E2 -792.4733} C_DIS
LIN {X -25.6868,Y 9.5209,Z 59,A 151.5041,B 24.8201,C -3.0932,E1 24.8506,E2 -788.7347} C_DIS
LIN {X -24.9515,Y 11.3085,Z 59,A 146.9269,B 24.8191,C -3.1019,E1 24.8557,E2 -784.1532} C_DIS
LIN {X -24.1643,Y 12.9056,Z 59,A 143.2663,B 24.8178,C -3.1129,E1 24.8604,E2 -780.4995} C_DIS
LIN {X -23.0244,Y 14.8441,Z 59,A 138.9758,B 24.816,C -3.1284,E1 24.8666,E2 -776.2241} C_DIS
LIN {X -22.131,Y 16.1458,Z 59,A 135.4126,B 24.8151,C -3.1356,E1 24.8724,E2 -772.6605} C_DIS
LIN {X -20.8908,Y 17.7212,Z 59,A 131.5442,B 24.8136,C -3.1483,E1 24.8792,E2 -768.8046} C_DIS
LIN {X -19.9854,Y 18.7364,Z 59,A 128.6745,B 24.8128,C -3.1551,E1 24.8846,E2 -765.9383} C_DIS
LIN {X -19.0859,Y 19.652,Z 59,A 125.4877,B 24.8125,C -3.158,E1 24.8909,E2 -762.7452} C_DIS
LIN {X -17.4118,Y 21.1492,Z 59,A 121.2626,B 24.8109,C -3.1714,E1 24.8998,E2 -758.5357} C_DIS
LIN {X -16.3181,Y 22.0046,Z 59,A 118.1059,B 24.8104,C -3.1756,E1 24.9068,E2 -755.3776} C_DIS
LIN {X -14.8946,Y 22.9916,Z 59,A 114.6942,B 24.8094,C -3.184,E1 24.9147,E2 -751.9745} C_DIS
LIN {X -13.742,Y 23.6988,Z 59,A 111.4753,B 24.8091,C -3.1862,E1 24.9224,E2 -748.7511} C_DIS
LIN {X -11.9795,Y 24.6363,Z 59,A 107.2422,B 24.8083,C -3.1924,E1 24.933,E2 -744.5214} C_DIS
LIN {X -9.9608,Y 25.5196,Z 59,A 103.0505,B 24.8072,C -3.2019,E1 24.9437,E2 -740.3428} C_DIS
LIN {X -8.3347,Y 26.0962,Z 59,A 99.098,B 24.807,C -3.2035,E1 24.9542,E2 -736.3867} C_DIS
LIN {X -6.8296,Y 26.5296,Z 59,A 95.9554,B 24.8065,C -3.2078,E1 24.9626,E2 -733.2496} C_DIS
LIN {X -5.1152,Y 26.9128,Z 59,A 92.2353,B 24.8062,C -3.2104,E1 24.9728,E2 -729.5315} C_DIS
LIN {X -3.4819,Y 27.1725,Z 59,A 88.734,B 24.8059,C -3.2123,E1 24.9825,E2 -726.0316} C_DIS
LIN {X -2.2725,Y 27.3004,Z 59,A 86.0113,B 24.8059,C -3.212,E1 24.9901,E2 -723.3069} C_DIS
LIN {X -0.5182,Y 27.3897,Z 59,A 82.6836,B 24.8055,C -3.216,E1 24.9993,E2 -719.9883} C_DIS
LIN {X 0.9935,Y 27.3766,Z 59,A 79.609,B 24.8053,C -3.2172,E1 25.0079,E2 -716.917} C_DIS
LIN {X 2.2517,Y 27.302,Z 59,A 76.0403,B 24.8064,C -3.2088,E1 25.0179,E2 -713.3301} C_DIS
LIN {X 5.414,Y 26.8542,Z 59,A 70.1969,B 24.8057,C -3.2144,E1 25.0339,E2 -707.5058} C_DIS
LIN {X 6.9751,Y 26.4917,Z 59,A 66.7783,B 24.806,C -3.2119,E1 25.0432,E2 -704.0863} C_DIS
LIN {X 8.2633,Y 26.1188,Z 59,A 63.9384,B 24.8063,C -3.2095,E1 25.0508,E2 -701.2458} C_DIS
LIN {X 10.4451,Y 25.3251,Z 59,A 58.8109,B 24.8071,C -3.2023,E1 25.0642,E2 -696.1123} C_DIS
Enddeposition()
END
